   1:  PR[GP1:91,1] = PR[GP1:90,1] + 38.057;
   1:  PR[GP1:91,2] = PR[GP1:90,2] + -35.573;
   1:L PR[91] 10mm/sec CNT100;
   1:  PR[GP1:91,1] = PR[GP1:90,1] + 42.822;
   1:  PR[GP1:91,2] = PR[GP1:90,2] + -33.695;
   1:L PR[91] 10mm/sec CNT100;
   1:  PR[GP1:91,1] = PR[GP1:90,1] + 46.775;
   1:  PR[GP1:91,2] = PR[GP1:90,2] + -32.295;
   1:L PR[91] 10mm/sec CNT100;
   1:  PR[GP1:91,1] = PR[GP1:90,1] + 51.154;
   1:  PR[GP1:91,2] = PR[GP1:90,2] + -29.580;
   1:L PR[91] 10mm/sec CNT100;
   1:  PR[GP1:91,1] = PR[GP1:90,1] + 55.415;
   1:  PR[GP1:91,2] = PR[GP1:90,2] + -25.807;
   1:L PR[91] 10mm/sec CNT100;
   1:  PR[GP1:91,1] = PR[GP1:90,1] + 57.463;
   1:  PR[GP1:91,2] = PR[GP1:90,2] + -24.149;
   1:L PR[91] 10mm/sec CNT100;
   1:  PR[GP1:91,1] = PR[GP1:90,1] + 60.946;
   1:  PR[GP1:91,2] = PR[GP1:90,2] + -19.628;
   1:L PR[91] 10mm/sec CNT100;
   1:  PR[GP1:91,1] = PR[GP1:90,1] + 63.849;
   1:  PR[GP1:91,2] = PR[GP1:90,2] + -14.057;
   1:L PR[91] 10mm/sec CNT100;
   1:  PR[GP1:91,1] = PR[GP1:90,1] + 64.641;
   1:  PR[GP1:91,2] = PR[GP1:90,2] + -12.738;
   1:L PR[91] 10mm/sec CNT100;
   1:  PR[GP1:91,1] = PR[GP1:90,1] + 66.291;
   1:  PR[GP1:91,2] = PR[GP1:90,2] + -7.215;
   1:L PR[91] 10mm/sec CNT100;
   1:  PR[GP1:91,1] = PR[GP1:90,1] + 66.863;
   1:  PR[GP1:91,2] = PR[GP1:90,2] + -1.098;
   1:L PR[91] 10mm/sec CNT100;
   1:  PR[GP1:91,1] = PR[GP1:90,1] + 67.069;
   1:  PR[GP1:91,2] = PR[GP1:90,2] + 0.023;
   1:L PR[91] 10mm/sec CNT100;
   1:  PR[GP1:91,1] = PR[GP1:90,1] + 66.517;
   1:  PR[GP1:91,2] = PR[GP1:90,2] + 6.002;
   1:L PR[91] 10mm/sec CNT100;
   1:  PR[GP1:91,1] = PR[GP1:90,1] + 66.299;
   1:  PR[GP1:91,2] = PR[GP1:90,2] + 7.180;
   1:L PR[91] 10mm/sec CNT100;
   1:  PR[GP1:91,1] = PR[GP1:90,1] + 64.636;
   1:  PR[GP1:91,2] = PR[GP1:90,2] + 12.747;
   1:L PR[91] 10mm/sec CNT100;
   1:  PR[GP1:91,1] = PR[GP1:90,1] + 61.933;
   1:  PR[GP1:91,2] = PR[GP1:90,2] + 17.984;
   1:L PR[91] 10mm/sec CNT100;
   1:  PR[GP1:91,1] = PR[GP1:90,1] + 60.958;
   1:  PR[GP1:91,2] = PR[GP1:90,2] + 19.603;
   1:L PR[91] 10mm/sec CNT100;
   1:  PR[GP1:91,1] = PR[GP1:90,1] + 57.455;
   1:  PR[GP1:91,2] = PR[GP1:90,2] + 24.151;
   1:L PR[91] 10mm/sec CNT100;
   1:  PR[GP1:91,1] = PR[GP1:90,1] + 53.581;
   1:  PR[GP1:91,2] = PR[GP1:90,2] + 27.615;
   1:L PR[91] 10mm/sec CNT100;
   1:  PR[GP1:91,1] = PR[GP1:90,1] + 51.169;
   1:  PR[GP1:91,2] = PR[GP1:90,2] + 29.562;
   1:L PR[91] 10mm/sec CNT100;
   1:  PR[GP1:91,1] = PR[GP1:90,1] + 46.768;
   1:  PR[GP1:91,2] = PR[GP1:90,2] + 32.290;
   1:L PR[91] 10mm/sec CNT100;
   1:  PR[GP1:91,1] = PR[GP1:90,1] + 42.433;
   1:  PR[GP1:91,2] = PR[GP1:90,2] + 34.022;
   1:L PR[91] 10mm/sec CNT100;
   1:  PR[GP1:91,1] = PR[GP1:90,1] + 38.074;
   1:  PR[GP1:91,2] = PR[GP1:90,2] + 35.561;
   1:L PR[91] 10mm/sec CNT100;
   1:  PR[GP1:91,1] = PR[GP1:90,1] + 33.724;
   1:  PR[GP1:91,2] = PR[GP1:90,2] + 36.497;
   1:L PR[91] 10mm/sec CNT100;
   1:  PR[GP1:91,1] = PR[GP1:90,1] + 29.795;
   1:  PR[GP1:91,2] = PR[GP1:90,2] + 36.645;
   1:L PR[91] 10mm/sec CNT100;
   1:  PR[GP1:91,1] = PR[GP1:90,1] + 23.624;
   1:  PR[GP1:91,2] = PR[GP1:90,2] + 36.667;
   1:L PR[91] 10mm/sec CNT100;
   1:  PR[GP1:91,1] = PR[GP1:90,1] + 20.005;
   1:  PR[GP1:91,2] = PR[GP1:90,2] + 36.191;
   1:L PR[91] 10mm/sec CNT100;
   1:  PR[GP1:91,1] = PR[GP1:90,1] + 16.894;
   1:  PR[GP1:91,2] = PR[GP1:90,2] + 35.201;
   1:L PR[91] 10mm/sec CNT100;
   1:  PR[GP1:91,1] = PR[GP1:90,1] + 9.875;
   1:  PR[GP1:91,2] = PR[GP1:90,2] + 32.768;
   1:L PR[91] 10mm/sec CNT100;
   1:  PR[GP1:91,1] = PR[GP1:90,1] + 7.298;
   1:  PR[GP1:91,2] = PR[GP1:90,2] + 31.423;
   1:L PR[91] 10mm/sec CNT100;
   1:  PR[GP1:91,1] = PR[GP1:90,1] + 3.973;
   1:  PR[GP1:91,2] = PR[GP1:90,2] + 29.074;
   1:L PR[91] 10mm/sec CNT100;
   1:  PR[GP1:91,1] = PR[GP1:90,1] + 3.823;
   1:  PR[GP1:91,2] = PR[GP1:90,2] + 28.957;
   1:L PR[91] 10mm/sec CNT100;
   1:  PR[GP1:91,1] = PR[GP1:90,1] + 3.611;
   1:  PR[GP1:91,2] = PR[GP1:90,2] + 28.710;
   1:L PR[91] 10mm/sec CNT100;
   1:  PR[GP1:91,1] = PR[GP1:90,1] + 2.937;
   1:  PR[GP1:91,2] = PR[GP1:90,2] + 28.444;
   1:L PR[91] 10mm/sec CNT100;
   1:  PR[GP1:91,1] = PR[GP1:90,1] + 1.783;
   1:  PR[GP1:91,2] = PR[GP1:90,2] + 27.801;
   1:L PR[91] 10mm/sec CNT100;
   1:  PR[GP1:91,1] = PR[GP1:90,1] + 0.780;
   1:  PR[GP1:91,2] = PR[GP1:90,2] + 28.419;
   1:  PR[GP1:91,3] = PR[GP1:90,3] + 58.520;
   1:L PR[91] 10mm/sec CNT100;
   1:  PR[GP1:91,1] = PR[GP1:90,1] + -2.625;
   1:  PR[GP1:91,2] = PR[GP1:90,2] + 29.211;
   1:L PR[91] 10mm/sec CNT100;
   1:  PR[GP1:91,1] = PR[GP1:90,1] + -6.013;
   1:  PR[GP1:91,2] = PR[GP1:90,2] + 31.605;
   1:L PR[91] 10mm/sec CNT100;
   1:  PR[GP1:91,1] = PR[GP1:90,1] + -8.315;
   1:  PR[GP1:91,2] = PR[GP1:90,2] + 32.809;
   1:L PR[91] 10mm/sec CNT100;
   1:  PR[GP1:91,1] = PR[GP1:90,1] + -11.164;
   1:  PR[GP1:91,2] = PR[GP1:90,2] + 33.725;
   1:L PR[91] 10mm/sec CNT100;
   1:  PR[GP1:91,1] = PR[GP1:90,1] + -18.764;
   1:  PR[GP1:91,2] = PR[GP1:90,2] + 36.352;
   1:L PR[91] 10mm/sec CNT100;
   1:  PR[GP1:91,1] = PR[GP1:90,1] + -22.038;
   1:  PR[GP1:91,2] = PR[GP1:90,2] + 36.780;
   1:L PR[91] 10mm/sec CNT100;
   1:  PR[GP1:91,1] = PR[GP1:90,1] + -25.898;
   1:  PR[GP1:91,2] = PR[GP1:90,2] + 36.647;
   1:L PR[91] 10mm/sec CNT100;
   1:  PR[GP1:91,1] = PR[GP1:90,1] + -32.531;
   1:  PR[GP1:91,2] = PR[GP1:90,2] + 36.614;
   1:L PR[91] 10mm/sec CNT100;
   1:  PR[GP1:91,1] = PR[GP1:90,1] + -36.524;
   1:  PR[GP1:91,2] = PR[GP1:90,2] + 35.753;
   1:L PR[91] 10mm/sec CNT100;
   1:  PR[GP1:91,1] = PR[GP1:90,1] + -40.912;
   1:  PR[GP1:91,2] = PR[GP1:90,2] + 34.015;
   1:L PR[91] 10mm/sec CNT100;
   1:  PR[GP1:91,1] = PR[GP1:90,1] + -45.583;
   1:  PR[GP1:91,2] = PR[GP1:90,2] + 32.357;
   1:L PR[91] 10mm/sec CNT100;
   1:  PR[GP1:91,1] = PR[GP1:90,1] + -49.681;
   1:  PR[GP1:91,2] = PR[GP1:90,2] + 29.804;
   1:L PR[91] 10mm/sec CNT100;
   1:  PR[GP1:91,1] = PR[GP1:90,1] + -53.670;
   1:  PR[GP1:91,2] = PR[GP1:90,2] + 26.262;
   1:L PR[91] 10mm/sec CNT100;
   1:  PR[GP1:91,1] = PR[GP1:90,1] + -56.314;
   1:  PR[GP1:91,2] = PR[GP1:90,2] + 24.122;
   1:L PR[91] 10mm/sec CNT100;
   1:  PR[GP1:91,1] = PR[GP1:90,1] + -59.540;
   1:  PR[GP1:91,2] = PR[GP1:90,2] + 19.923;
   1:L PR[91] 10mm/sec CNT100;
   1:  PR[GP1:91,1] = PR[GP1:90,1] + -62.253;
   1:  PR[GP1:91,2] = PR[GP1:90,2] + 14.659;
   1:L PR[91] 10mm/sec CNT100;
   1:  PR[GP1:91,1] = PR[GP1:90,1] + -63.437;
   1:  PR[GP1:91,2] = PR[GP1:90,2] + 12.681;
   1:L PR[91] 10mm/sec CNT100;
   1:  PR[GP1:91,1] = PR[GP1:90,1] + -64.989;
   1:  PR[GP1:91,2] = PR[GP1:90,2] + 7.415;
   1:L PR[91] 10mm/sec CNT100;
   1:  PR[GP1:91,1] = PR[GP1:90,1] + -65.501;
   1:  PR[GP1:91,2] = PR[GP1:90,2] + 1.817;
   1:L PR[91] 10mm/sec CNT100;
   1:  PR[GP1:91,1] = PR[GP1:90,1] + -65.842;
   1:  PR[GP1:91,2] = PR[GP1:90,2] + -0.032;
   1:L PR[91] 10mm/sec CNT100;
   1:  PR[GP1:91,1] = PR[GP1:90,1] + -65.348;
   1:  PR[GP1:91,2] = PR[GP1:90,2] + -5.509;
   1:L PR[91] 10mm/sec CNT100;
   1:  PR[GP1:91,1] = PR[GP1:90,1] + -64.997;
   1:  PR[GP1:91,2] = PR[GP1:90,2] + -7.398;
   1:L PR[91] 10mm/sec CNT100;
   1:  PR[GP1:91,1] = PR[GP1:90,1] + -63.431;
   1:  PR[GP1:91,2] = PR[GP1:90,2] + -12.710;
   1:L PR[91] 10mm/sec CNT100;
   1:  PR[GP1:91,1] = PR[GP1:90,1] + -60.899;
   1:  PR[GP1:91,2] = PR[GP1:90,2] + -17.675;
   1:L PR[91] 10mm/sec CNT100;
   1:  PR[GP1:91,1] = PR[GP1:90,1] + -59.551;
   1:  PR[GP1:91,2] = PR[GP1:90,2] + -19.917;
   1:L PR[91] 10mm/sec CNT100;
   1:  PR[GP1:91,1] = PR[GP1:90,1] + -56.303;
   1:  PR[GP1:91,2] = PR[GP1:90,2] + -24.145;
   1:L PR[91] 10mm/sec CNT100;
   1:  PR[GP1:91,1] = PR[GP1:90,1] + -52.655;
   1:  PR[GP1:91,2] = PR[GP1:90,2] + -27.417;
   1:L PR[91] 10mm/sec CNT100;
   1:  PR[GP1:91,1] = PR[GP1:90,1] + -49.690;
   1:  PR[GP1:91,2] = PR[GP1:90,2] + -29.807;
   1:L PR[91] 10mm/sec CNT100;
   1:  PR[GP1:91,1] = PR[GP1:90,1] + -45.569;
   1:  PR[GP1:91,2] = PR[GP1:90,2] + -32.374;
   1:L PR[91] 10mm/sec CNT100;
   1:  PR[GP1:91,1] = PR[GP1:90,1] + -41.541;
   1:  PR[GP1:91,2] = PR[GP1:90,2] + -33.992;
   1:L PR[91] 10mm/sec CNT100;
   1:  PR[GP1:91,1] = PR[GP1:90,1] + -36.528;
   1:  PR[GP1:91,2] = PR[GP1:90,2] + -35.760;
   1:L PR[91] 10mm/sec CNT100;
   1:  PR[GP1:91,1] = PR[GP1:90,1] + -32.514;
   1:  PR[GP1:91,2] = PR[GP1:90,2] + -36.626;
   1:L PR[91] 10mm/sec CNT100;
   1:  PR[GP1:91,1] = PR[GP1:90,1] + -28.876;
   1:  PR[GP1:91,2] = PR[GP1:90,2] + -36.766;
   1:L PR[91] 10mm/sec CNT100;
   1:  PR[GP1:91,1] = PR[GP1:90,1] + -22.036;
   1:  PR[GP1:91,2] = PR[GP1:90,2] + -36.788;
   1:L PR[91] 10mm/sec CNT100;
   1:  PR[GP1:91,1] = PR[GP1:90,1] + -18.744;
   1:  PR[GP1:91,2] = PR[GP1:90,2] + -36.358;
   1:L PR[91] 10mm/sec CNT100;
   1:  PR[GP1:91,1] = PR[GP1:90,1] + -15.922;
   1:  PR[GP1:91,2] = PR[GP1:90,2] + -35.460;
   1:L PR[91] 10mm/sec CNT100;
   1:  PR[GP1:91,1] = PR[GP1:90,1] + -8.309;
   1:  PR[GP1:91,2] = PR[GP1:90,2] + -32.814;
   1:L PR[91] 10mm/sec CNT100;
   1:  PR[GP1:91,1] = PR[GP1:90,1] + -6.009;
   1:  PR[GP1:91,2] = PR[GP1:90,2] + -31.611;
   1:L PR[91] 10mm/sec CNT100;
   1:  PR[GP1:91,1] = PR[GP1:90,1] + -2.582;
   1:  PR[GP1:91,2] = PR[GP1:90,2] + -29.121;
   1:L PR[91] 10mm/sec CNT100;
   1:  PR[GP1:91,1] = PR[GP1:90,1] + -1.792;
   1:  PR[GP1:91,2] = PR[GP1:90,2] + -29.090;
   1:L PR[91] 10mm/sec CNT100;
   1:  PR[GP1:91,1] = PR[GP1:90,1] + 1.871;
   1:  PR[GP1:91,2] = PR[GP1:90,2] + -28.308;
   1:L PR[91] 10mm/sec CNT100;
   1:  PR[GP1:91,1] = PR[GP1:90,1] + 2.128;
   1:  PR[GP1:91,2] = PR[GP1:90,2] + -28.515;
   1:L PR[91] 10mm/sec CNT100;
   1:  PR[GP1:91,1] = PR[GP1:90,1] + 3.505;
   1:  PR[GP1:91,2] = PR[GP1:90,2] + -29.200;
   1:L PR[91] 10mm/sec CNT100;
   1:  PR[GP1:91,1] = PR[GP1:90,1] + 6.833;
   1:  PR[GP1:91,2] = PR[GP1:90,2] + -31.618;
   1:L PR[91] 10mm/sec CNT100;
   1:  PR[GP1:91,1] = PR[GP1:90,1] + 9.111;
   1:  PR[GP1:91,2] = PR[GP1:90,2] + -32.807;
   1:L PR[91] 10mm/sec CNT100;
   1:  PR[GP1:91,1] = PR[GP1:90,1] + 11.958;
   1:  PR[GP1:91,2] = PR[GP1:90,2] + -33.722;
   1:L PR[91] 10mm/sec CNT100;
   1:  PR[GP1:91,1] = PR[GP1:90,1] + 19.568;
   1:  PR[GP1:91,2] = PR[GP1:90,2] + -36.356;
   1:L PR[91] 10mm/sec CNT100;
   1:  PR[GP1:91,1] = PR[GP1:90,1] + 22.838;
   1:  PR[GP1:91,2] = PR[GP1:90,2] + -36.786;
   1:L PR[91] 10mm/sec CNT100;
   1:  PR[GP1:91,1] = PR[GP1:90,1] + 26.679;
   1:  PR[GP1:91,2] = PR[GP1:90,2] + -36.657;
   1:L PR[91] 10mm/sec CNT100;
   1:  PR[GP1:91,1] = PR[GP1:90,1] + 33.319;
   1:  PR[GP1:91,2] = PR[GP1:90,2] + -36.628;
   1:L PR[91] 10mm/sec CNT100;
   1:  PR[GP1:91,1] = PR[GP1:90,1] + 37.305;
   1:  PR[GP1:91,2] = PR[GP1:90,2] + -35.770;
   1:L PR[91] 10mm/sec CNT100;
   1:  PR[GP1:91,1] = PR[GP1:90,1] + 41.699;
   1:  PR[GP1:91,2] = PR[GP1:90,2] + -34.039;
   1:L PR[91] 10mm/sec CNT100;
   1:  PR[GP1:91,1] = PR[GP1:90,1] + 46.376;
   1:  PR[GP1:91,2] = PR[GP1:90,2] + -32.381;
   1:L PR[91] 10mm/sec CNT100;
   1:  PR[GP1:91,1] = PR[GP1:90,1] + 50.449;
   1:  PR[GP1:91,2] = PR[GP1:90,2] + -29.857;
   1:L PR[91] 10mm/sec CNT100;
   1:  PR[GP1:91,1] = PR[GP1:90,1] + 54.416;
   1:  PR[GP1:91,2] = PR[GP1:90,2] + -26.344;
   1:L PR[91] 10mm/sec CNT100;
   1:  PR[GP1:91,1] = PR[GP1:90,1] + 57.067;
   1:  PR[GP1:91,2] = PR[GP1:90,2] + -24.198;
   1:L PR[91] 10mm/sec CNT100;
   1:  PR[GP1:91,1] = PR[GP1:90,1] + 60.327;
   1:  PR[GP1:91,2] = PR[GP1:90,2] + -19.966;
   1:L PR[91] 10mm/sec CNT100;
   1:  PR[GP1:91,1] = PR[GP1:90,1] + 63.048;
   1:  PR[GP1:91,2] = PR[GP1:90,2] + -14.745;
   1:L PR[91] 10mm/sec CNT100;
   1:  PR[GP1:91,1] = PR[GP1:90,1] + 64.235;
   1:  PR[GP1:91,2] = PR[GP1:90,2] + -12.768;
   1:L PR[91] 10mm/sec CNT100;
   1:  PR[GP1:91,1] = PR[GP1:90,1] + 65.784;
   1:  PR[GP1:91,2] = PR[GP1:90,2] + -7.581;
   1:L PR[91] 10mm/sec CNT100;
   1:  PR[GP1:91,1] = PR[GP1:90,1] + 66.322;
   1:  PR[GP1:91,2] = PR[GP1:90,2] + -1.828;
   1:L PR[91] 10mm/sec CNT100;
   1:  PR[GP1:91,1] = PR[GP1:90,1] + 66.663;
   1:  PR[GP1:91,2] = PR[GP1:90,2] + 0.023;
   1:L PR[91] 10mm/sec CNT100;
   1:  PR[GP1:91,1] = PR[GP1:90,1] + 66.143;
   1:  PR[GP1:91,2] = PR[GP1:90,2] + 5.652;
   1:L PR[91] 10mm/sec CNT100;
   1:  PR[GP1:91,1] = PR[GP1:90,1] + 65.792;
   1:  PR[GP1:91,2] = PR[GP1:90,2] + 7.545;
   1:L PR[91] 10mm/sec CNT100;
   1:  PR[GP1:91,1] = PR[GP1:90,1] + 64.229;
   1:  PR[GP1:91,2] = PR[GP1:90,2] + 12.777;
   1:L PR[91] 10mm/sec CNT100;
   1:  PR[GP1:91,1] = PR[GP1:90,1] + 61.689;
   1:  PR[GP1:91,2] = PR[GP1:90,2] + 17.700;
   1:L PR[91] 10mm/sec CNT100;
   1:  PR[GP1:91,1] = PR[GP1:90,1] + 60.340;
   1:  PR[GP1:91,2] = PR[GP1:90,2] + 19.941;
   1:L PR[91] 10mm/sec CNT100;
   1:  PR[GP1:91,1] = PR[GP1:90,1] + 57.060;
   1:  PR[GP1:91,2] = PR[GP1:90,2] + 24.199;
   1:L PR[91] 10mm/sec CNT100;
   1:  PR[GP1:91,1] = PR[GP1:90,1] + 53.431;
   1:  PR[GP1:91,2] = PR[GP1:90,2] + 27.444;
   1:L PR[91] 10mm/sec CNT100;
   1:  PR[GP1:91,1] = PR[GP1:90,1] + 50.464;
   1:  PR[GP1:91,2] = PR[GP1:90,2] + 29.839;
   1:L PR[91] 10mm/sec CNT100;
   1:  PR[GP1:91,1] = PR[GP1:90,1] + 46.370;
   1:  PR[GP1:91,2] = PR[GP1:90,2] + 32.377;
   1:L PR[91] 10mm/sec CNT100;
   1:  PR[GP1:91,1] = PR[GP1:90,1] + 42.336;
   1:  PR[GP1:91,2] = PR[GP1:90,2] + 33.988;
   1:L PR[91] 10mm/sec CNT100;
   1:  PR[GP1:91,1] = PR[GP1:90,1] + 37.323;
   1:  PR[GP1:91,2] = PR[GP1:90,2] + 35.758;
   1:L PR[91] 10mm/sec CNT100;
   1:  PR[GP1:91,1] = PR[GP1:90,1] + 33.316;
   1:  PR[GP1:91,2] = PR[GP1:90,2] + 36.620;
   1:L PR[91] 10mm/sec CNT100;
   1:  PR[GP1:91,1] = PR[GP1:90,1] + 29.696;
   1:  PR[GP1:91,2] = PR[GP1:90,2] + 36.757;
   1:L PR[91] 10mm/sec CNT100;
   1:  PR[GP1:91,1] = PR[GP1:90,1] + 22.858;
   1:  PR[GP1:91,2] = PR[GP1:90,2] + 36.781;
   1:L PR[91] 10mm/sec CNT100;
   1:  PR[GP1:91,1] = PR[GP1:90,1] + 19.572;
   1:  PR[GP1:91,2] = PR[GP1:90,2] + 36.349;
   1:L PR[91] 10mm/sec CNT100;
   1:  PR[GP1:91,1] = PR[GP1:90,1] + 16.746;
   1:  PR[GP1:91,2] = PR[GP1:90,2] + 35.449;
   1:L PR[91] 10mm/sec CNT100;
   1:  PR[GP1:91,1] = PR[GP1:90,1] + 9.130;
   1:  PR[GP1:91,2] = PR[GP1:90,2] + 32.809;
   1:L PR[91] 10mm/sec CNT100;
   1:  PR[GP1:91,1] = PR[GP1:90,1] + 6.837;
   1:  PR[GP1:91,2] = PR[GP1:90,2] + 31.612;
   1:L PR[91] 10mm/sec CNT100;
   1:  PR[GP1:91,1] = PR[GP1:90,1] + 3.510;
   1:  PR[GP1:91,2] = PR[GP1:90,2] + 29.256;
   1:L PR[91] 10mm/sec CNT100;
   1:  PR[GP1:91,1] = PR[GP1:90,1] + 1.849;
   1:  PR[GP1:91,2] = PR[GP1:90,2] + 28.332;
   1:L PR[91] 10mm/sec CNT100;
   1:  PR[GP1:91,1] = PR[GP1:90,1] + 0.451;
   1:  PR[GP1:91,2] = PR[GP1:90,2] + 28.982;
   1:  PR[GP1:91,3] = PR[GP1:90,3] + 59.850;
   1:L PR[91] 10mm/sec CNT100;
   1:  PR[GP1:91,1] = PR[GP1:90,1] + -2.564;
   1:  PR[GP1:91,2] = PR[GP1:90,2] + 29.683;
   1:L PR[91] 10mm/sec CNT100;
   1:  PR[GP1:91,1] = PR[GP1:90,1] + -5.554;
   1:  PR[GP1:91,2] = PR[GP1:90,2] + 31.796;
   1:L PR[91] 10mm/sec CNT100;
   1:  PR[GP1:91,1] = PR[GP1:90,1] + -7.570;
   1:  PR[GP1:91,2] = PR[GP1:90,2] + 32.850;
   1:L PR[91] 10mm/sec CNT100;
   1:  PR[GP1:91,1] = PR[GP1:90,1] + -10.072;
   1:  PR[GP1:91,2] = PR[GP1:90,2] + 33.654;
   1:L PR[91] 10mm/sec CNT100;
   1:  PR[GP1:91,1] = PR[GP1:90,1] + -18.331;
   1:  PR[GP1:91,2] = PR[GP1:90,2] + 36.509;
   1:L PR[91] 10mm/sec CNT100;
   1:  PR[GP1:91,1] = PR[GP1:90,1] + -21.272;
   1:  PR[GP1:91,2] = PR[GP1:90,2] + 36.894;
   1:L PR[91] 10mm/sec CNT100;
   1:  PR[GP1:91,1] = PR[GP1:90,1] + -24.746;
   1:  PR[GP1:91,2] = PR[GP1:90,2] + 36.774;
   1:L PR[91] 10mm/sec CNT100;
   1:  PR[GP1:91,1] = PR[GP1:90,1] + -32.122;
   1:  PR[GP1:91,2] = PR[GP1:90,2] + 36.737;
   1:L PR[91] 10mm/sec CNT100;
   1:  PR[GP1:91,1] = PR[GP1:90,1] + -35.770;
   1:  PR[GP1:91,2] = PR[GP1:90,2] + 35.950;
   1:L PR[91] 10mm/sec CNT100;
   1:  PR[GP1:91,1] = PR[GP1:90,1] + -39.787;
   1:  PR[GP1:91,2] = PR[GP1:90,2] + 34.360;
   1:L PR[91] 10mm/sec CNT100;
   1:  PR[GP1:91,1] = PR[GP1:90,1] + -45.183;
   1:  PR[GP1:91,2] = PR[GP1:90,2] + 32.444;
   1:L PR[91] 10mm/sec CNT100;
   1:  PR[GP1:91,1] = PR[GP1:90,1] + -48.972;
   1:  PR[GP1:91,2] = PR[GP1:90,2] + 30.083;
   1:L PR[91] 10mm/sec CNT100;
   1:  PR[GP1:91,1] = PR[GP1:90,1] + -52.666;
   1:  PR[GP1:91,2] = PR[GP1:90,2] + 26.803;
   1:L PR[91] 10mm/sec CNT100;
   1:  PR[GP1:91,1] = PR[GP1:90,1] + -55.914;
   1:  PR[GP1:91,2] = PR[GP1:90,2] + 24.175;
   1:L PR[91] 10mm/sec CNT100;
   1:  PR[GP1:91,1] = PR[GP1:90,1] + -58.920;
   1:  PR[GP1:91,2] = PR[GP1:90,2] + 20.263;
   1:L PR[91] 10mm/sec CNT100;
   1:  PR[GP1:91,1] = PR[GP1:90,1] + -61.450;
   1:  PR[GP1:91,2] = PR[GP1:90,2] + 15.353;
   1:L PR[91] 10mm/sec CNT100;
   1:  PR[GP1:91,1] = PR[GP1:90,1] + -63.029;
   1:  PR[GP1:91,2] = PR[GP1:90,2] + 12.715;
   1:L PR[91] 10mm/sec CNT100;
   1:  PR[GP1:91,1] = PR[GP1:90,1] + -64.481;
   1:  PR[GP1:91,2] = PR[GP1:90,2] + 7.789;
   1:L PR[91] 10mm/sec CNT100;
   1:  PR[GP1:91,1] = PR[GP1:90,1] + -64.961;
   1:  PR[GP1:91,2] = PR[GP1:90,2] + 2.546;
   1:L PR[91] 10mm/sec CNT100;
   1:  PR[GP1:91,1] = PR[GP1:90,1] + -65.436;
   1:  PR[GP1:91,2] = PR[GP1:90,2] + -0.032;
   1:L PR[91] 10mm/sec CNT100;
   1:  PR[GP1:91,1] = PR[GP1:90,1] + -64.972;
   1:  PR[GP1:91,2] = PR[GP1:90,2] + -5.168;
   1:L PR[91] 10mm/sec CNT100;
   1:  PR[GP1:91,1] = PR[GP1:90,1] + -64.489;
   1:  PR[GP1:91,2] = PR[GP1:90,2] + -7.772;
   1:L PR[91] 10mm/sec CNT100;
   1:  PR[GP1:91,1] = PR[GP1:90,1] + -63.023;
   1:  PR[GP1:91,2] = PR[GP1:90,2] + -12.744;
   1:L PR[91] 10mm/sec CNT100;
   1:  PR[GP1:91,1] = PR[GP1:90,1] + -60.652;
   1:  PR[GP1:91,2] = PR[GP1:90,2] + -17.392;
   1:L PR[91] 10mm/sec CNT100;
   1:  PR[GP1:91,1] = PR[GP1:90,1] + -58.930;
   1:  PR[GP1:91,2] = PR[GP1:90,2] + -20.258;
   1:L PR[91] 10mm/sec CNT100;
   1:  PR[GP1:91,1] = PR[GP1:90,1] + -55.903;
   1:  PR[GP1:91,2] = PR[GP1:90,2] + -24.198;
   1:L PR[91] 10mm/sec CNT100;
   1:  PR[GP1:91,1] = PR[GP1:90,1] + -52.502;
   1:  PR[GP1:91,2] = PR[GP1:90,2] + -27.248;
   1:L PR[91] 10mm/sec CNT100;
   1:  PR[GP1:91,1] = PR[GP1:90,1] + -48.981;
   1:  PR[GP1:91,2] = PR[GP1:90,2] + -30.087;
   1:L PR[91] 10mm/sec CNT100;
   1:  PR[GP1:91,1] = PR[GP1:90,1] + -45.168;
   1:  PR[GP1:91,2] = PR[GP1:90,2] + -32.462;
   1:L PR[91] 10mm/sec CNT100;
   1:  PR[GP1:91,1] = PR[GP1:90,1] + -41.441;
   1:  PR[GP1:91,2] = PR[GP1:90,2] + -33.959;
   1:L PR[91] 10mm/sec CNT100;
   1:  PR[GP1:91,1] = PR[GP1:90,1] + -35.773;
   1:  PR[GP1:91,2] = PR[GP1:90,2] + -35.958;
   1:L PR[91] 10mm/sec CNT100;
   1:  PR[GP1:91,1] = PR[GP1:90,1] + -32.104;
   1:  PR[GP1:91,2] = PR[GP1:90,2] + -36.750;
   1:L PR[91] 10mm/sec CNT100;
   1:  PR[GP1:91,1] = PR[GP1:90,1] + -28.776;
   1:  PR[GP1:91,2] = PR[GP1:90,2] + -36.878;
   1:L PR[91] 10mm/sec CNT100;
   1:  PR[GP1:91,1] = PR[GP1:90,1] + -21.268;
   1:  PR[GP1:91,2] = PR[GP1:90,2] + -36.902;
   1:L PR[91] 10mm/sec CNT100;
   1:  PR[GP1:91,1] = PR[GP1:90,1] + -18.311;
   1:  PR[GP1:91,2] = PR[GP1:90,2] + -36.515;
   1:L PR[91] 10mm/sec CNT100;
   1:  PR[GP1:91,1] = PR[GP1:90,1] + -15.773;
   1:  PR[GP1:91,2] = PR[GP1:90,2] + -35.708;
   1:L PR[91] 10mm/sec CNT100;
   1:  PR[GP1:91,1] = PR[GP1:90,1] + -7.563;
   1:  PR[GP1:91,2] = PR[GP1:90,2] + -32.854;
   1:L PR[91] 10mm/sec CNT100;
   1:  PR[GP1:91,1] = PR[GP1:90,1] + -5.549;
   1:  PR[GP1:91,2] = PR[GP1:90,2] + -31.801;
   1:L PR[91] 10mm/sec CNT100;
   1:  PR[GP1:91,1] = PR[GP1:90,1] + -2.522;
   1:  PR[GP1:91,2] = PR[GP1:90,2] + -29.602;
   1:L PR[91] 10mm/sec CNT100;
   1:  PR[GP1:91,1] = PR[GP1:90,1] + -1.431;
   1:  PR[GP1:91,2] = PR[GP1:90,2] + -29.558;
   1:L PR[91] 10mm/sec CNT100;
   1:  PR[GP1:91,1] = PR[GP1:90,1] + 1.938;
   1:  PR[GP1:91,2] = PR[GP1:90,2] + -28.839;
   1:L PR[91] 10mm/sec CNT100;
   1:  PR[GP1:91,1] = PR[GP1:90,1] + 2.234;
   1:  PR[GP1:91,2] = PR[GP1:90,2] + -29.078;
   1:L PR[91] 10mm/sec CNT100;
   1:  PR[GP1:91,1] = PR[GP1:90,1] + 3.443;
   1:  PR[GP1:91,2] = PR[GP1:90,2] + -29.680;
   1:L PR[91] 10mm/sec CNT100;
   1:  PR[GP1:91,1] = PR[GP1:90,1] + 6.371;
   1:  PR[GP1:91,2] = PR[GP1:90,2] + -31.807;
   1:L PR[91] 10mm/sec CNT100;
   1:  PR[GP1:91,1] = PR[GP1:90,1] + 8.365;
   1:  PR[GP1:91,2] = PR[GP1:90,2] + -32.848;
   1:L PR[91] 10mm/sec CNT100;
   1:  PR[GP1:91,1] = PR[GP1:90,1] + 10.864;
   1:  PR[GP1:91,2] = PR[GP1:90,2] + -33.651;
   1:L PR[91] 10mm/sec CNT100;
   1:  PR[GP1:91,1] = PR[GP1:90,1] + 19.135;
   1:  PR[GP1:91,2] = PR[GP1:90,2] + -36.514;
   1:L PR[91] 10mm/sec CNT100;
   1:  PR[GP1:91,1] = PR[GP1:90,1] + 22.071;
   1:  PR[GP1:91,2] = PR[GP1:90,2] + -36.900;
   1:L PR[91] 10mm/sec CNT100;
   1:  PR[GP1:91,1] = PR[GP1:90,1] + 25.529;
   1:  PR[GP1:91,2] = PR[GP1:90,2] + -36.784;
   1:L PR[91] 10mm/sec CNT100;
   1:  PR[GP1:91,1] = PR[GP1:90,1] + 32.910;
   1:  PR[GP1:91,2] = PR[GP1:90,2] + -36.751;
   1:L PR[91] 10mm/sec CNT100;
   1:  PR[GP1:91,1] = PR[GP1:90,1] + 36.553;
   1:  PR[GP1:91,2] = PR[GP1:90,2] + -35.967;
   1:L PR[91] 10mm/sec CNT100;
   1:  PR[GP1:91,1] = PR[GP1:90,1] + 40.575;
   1:  PR[GP1:91,2] = PR[GP1:90,2] + -34.383;
   1:L PR[91] 10mm/sec CNT100;
   1:  PR[GP1:91,1] = PR[GP1:90,1] + 45.977;
   1:  PR[GP1:91,2] = PR[GP1:90,2] + -32.468;
   1:L PR[91] 10mm/sec CNT100;
   1:  PR[GP1:91,1] = PR[GP1:90,1] + 49.743;
   1:  PR[GP1:91,2] = PR[GP1:90,2] + -30.134;
   1:L PR[91] 10mm/sec CNT100;
   1:  PR[GP1:91,1] = PR[GP1:90,1] + 53.416;
   1:  PR[GP1:91,2] = PR[GP1:90,2] + -26.881;
   1:L PR[91] 10mm/sec CNT100;
   1:  PR[GP1:91,1] = PR[GP1:90,1] + 56.671;
   1:  PR[GP1:91,2] = PR[GP1:90,2] + -24.246;
   1:L PR[91] 10mm/sec CNT100;
   1:  PR[GP1:91,1] = PR[GP1:90,1] + 59.709;
   1:  PR[GP1:91,2] = PR[GP1:90,2] + -20.303;
   1:L PR[91] 10mm/sec CNT100;
   1:  PR[GP1:91,1] = PR[GP1:90,1] + 62.246;
   1:  PR[GP1:91,2] = PR[GP1:90,2] + -15.434;
   1:L PR[91] 10mm/sec CNT100;
   1:  PR[GP1:91,1] = PR[GP1:90,1] + 63.828;
   1:  PR[GP1:91,2] = PR[GP1:90,2] + -12.799;
   1:L PR[91] 10mm/sec CNT100;
   1:  PR[GP1:91,1] = PR[GP1:90,1] + 65.278;
   1:  PR[GP1:91,2] = PR[GP1:90,2] + -7.946;
   1:L PR[91] 10mm/sec CNT100;
   1:  PR[GP1:91,1] = PR[GP1:90,1] + 65.781;
   1:  PR[GP1:91,2] = PR[GP1:90,2] + -2.558;
   1:L PR[91] 10mm/sec CNT100;
   1:  PR[GP1:91,1] = PR[GP1:90,1] + 66.257;
   1:  PR[GP1:91,2] = PR[GP1:90,2] + 0.023;
   1:L PR[91] 10mm/sec CNT100;
   1:  PR[GP1:91,1] = PR[GP1:90,1] + 65.769;
   1:  PR[GP1:91,2] = PR[GP1:90,2] + 5.301;
   1:L PR[91] 10mm/sec CNT100;
   1:  PR[GP1:91,1] = PR[GP1:90,1] + 65.286;
   1:  PR[GP1:91,2] = PR[GP1:90,2] + 7.911;
   1:L PR[91] 10mm/sec CNT100;
   1:  PR[GP1:91,1] = PR[GP1:90,1] + 63.823;
   1:  PR[GP1:91,2] = PR[GP1:90,2] + 12.808;
   1:L PR[91] 10mm/sec CNT100;
   1:  PR[GP1:91,1] = PR[GP1:90,1] + 61.445;
   1:  PR[GP1:91,2] = PR[GP1:90,2] + 17.415;
   1:L PR[91] 10mm/sec CNT100;
   1:  PR[GP1:91,1] = PR[GP1:90,1] + 59.722;
   1:  PR[GP1:91,2] = PR[GP1:90,2] + 20.278;
   1:L PR[91] 10mm/sec CNT100;
   1:  PR[GP1:91,1] = PR[GP1:90,1] + 56.664;
   1:  PR[GP1:91,2] = PR[GP1:90,2] + 24.247;
   1:L PR[91] 10mm/sec CNT100;
   1:  PR[GP1:91,1] = PR[GP1:90,1] + 53.282;
   1:  PR[GP1:91,2] = PR[GP1:90,2] + 27.272;
   1:L PR[91] 10mm/sec CNT100;
   1:  PR[GP1:91,1] = PR[GP1:90,1] + 49.759;
   1:  PR[GP1:91,2] = PR[GP1:90,2] + 30.116;
   1:L PR[91] 10mm/sec CNT100;
   1:  PR[GP1:91,1] = PR[GP1:90,1] + 45.971;
   1:  PR[GP1:91,2] = PR[GP1:90,2] + 32.463;
   1:L PR[91] 10mm/sec CNT100;
   1:  PR[GP1:91,1] = PR[GP1:90,1] + 42.239;
   1:  PR[GP1:91,2] = PR[GP1:90,2] + 33.954;
   1:L PR[91] 10mm/sec CNT100;
   1:  PR[GP1:91,1] = PR[GP1:90,1] + 36.572;
   1:  PR[GP1:91,2] = PR[GP1:90,2] + 35.955;
   1:L PR[91] 10mm/sec CNT100;
   1:  PR[GP1:91,1] = PR[GP1:90,1] + 32.909;
   1:  PR[GP1:91,2] = PR[GP1:90,2] + 36.743;
   1:L PR[91] 10mm/sec CNT100;
   1:  PR[GP1:91,1] = PR[GP1:90,1] + 29.598;
   1:  PR[GP1:91,2] = PR[GP1:90,2] + 36.868;
   1:L PR[91] 10mm/sec CNT100;
   1:  PR[GP1:91,1] = PR[GP1:90,1] + 22.092;
   1:  PR[GP1:91,2] = PR[GP1:90,2] + 36.894;
   1:L PR[91] 10mm/sec CNT100;
   1:  PR[GP1:91,1] = PR[GP1:90,1] + 19.140;
   1:  PR[GP1:91,2] = PR[GP1:90,2] + 36.506;
   1:L PR[91] 10mm/sec CNT100;
   1:  PR[GP1:91,1] = PR[GP1:90,1] + 16.598;
   1:  PR[GP1:91,2] = PR[GP1:90,2] + 35.698;
   1:L PR[91] 10mm/sec CNT100;
   1:  PR[GP1:91,1] = PR[GP1:90,1] + 8.385;
   1:  PR[GP1:91,2] = PR[GP1:90,2] + 32.850;
   1:L PR[91] 10mm/sec CNT100;
   1:  PR[GP1:91,1] = PR[GP1:90,1] + 6.376;
   1:  PR[GP1:91,2] = PR[GP1:90,2] + 31.802;
   1:L PR[91] 10mm/sec CNT100;
   1:  PR[GP1:91,1] = PR[GP1:90,1] + 3.745;
   1:  PR[GP1:91,2] = PR[GP1:90,2] + 29.943;
   1:L PR[91] 10mm/sec CNT100;
   1:  PR[GP1:91,1] = PR[GP1:90,1] + 3.748;
   1:  PR[GP1:91,2] = PR[GP1:90,2] + 29.883;
   1:L PR[91] 10mm/sec CNT100;
   1:  PR[GP1:91,1] = PR[GP1:90,1] + 1.914;
   1:  PR[GP1:91,2] = PR[GP1:90,2] + 28.862;
   1:L PR[91] 10mm/sec CNT100;
   1:  PR[GP1:91,1] = PR[GP1:90,1] + 0.122;
   1:  PR[GP1:91,2] = PR[GP1:90,2] + 29.545;
   1:  PR[GP1:91,3] = PR[GP1:90,3] + 61.180;
   1:L PR[91] 10mm/sec CNT100;
   1:  PR[GP1:91,1] = PR[GP1:90,1] + -2.504;
   1:  PR[GP1:91,2] = PR[GP1:90,2] + 30.155;
   1:L PR[91] 10mm/sec CNT100;
   1:  PR[GP1:91,1] = PR[GP1:90,1] + -5.095;
   1:  PR[GP1:91,2] = PR[GP1:90,2] + 31.986;
   1:L PR[91] 10mm/sec CNT100;
   1:  PR[GP1:91,1] = PR[GP1:90,1] + -6.825;
   1:  PR[GP1:91,2] = PR[GP1:90,2] + 32.891;
   1:L PR[91] 10mm/sec CNT100;
   1:  PR[GP1:91,1] = PR[GP1:90,1] + -8.980;
   1:  PR[GP1:91,2] = PR[GP1:90,2] + 33.584;
   1:L PR[91] 10mm/sec CNT100;
   1:  PR[GP1:91,1] = PR[GP1:90,1] + -17.898;
   1:  PR[GP1:91,2] = PR[GP1:90,2] + 36.667;
   1:L PR[91] 10mm/sec CNT100;
   1:  PR[GP1:91,1] = PR[GP1:90,1] + -20.505;
   1:  PR[GP1:91,2] = PR[GP1:90,2] + 37.008;
   1:L PR[91] 10mm/sec CNT100;
   1:  PR[GP1:91,1] = PR[GP1:90,1] + -23.595;
   1:  PR[GP1:91,2] = PR[GP1:90,2] + 36.901;
   1:L PR[91] 10mm/sec CNT100;
   1:  PR[GP1:91,1] = PR[GP1:90,1] + -31.713;
   1:  PR[GP1:91,2] = PR[GP1:90,2] + 36.861;
   1:L PR[91] 10mm/sec CNT100;
   1:  PR[GP1:91,1] = PR[GP1:90,1] + -35.017;
   1:  PR[GP1:91,2] = PR[GP1:90,2] + 36.148;
   1:L PR[91] 10mm/sec CNT100;
   1:  PR[GP1:91,1] = PR[GP1:90,1] + -38.662;
   1:  PR[GP1:91,2] = PR[GP1:90,2] + 34.705;
   1:L PR[91] 10mm/sec CNT100;
   1:  PR[GP1:91,1] = PR[GP1:90,1] + -44.783;
   1:  PR[GP1:91,2] = PR[GP1:90,2] + 32.531;
   1:L PR[91] 10mm/sec CNT100;
   1:  PR[GP1:91,1] = PR[GP1:90,1] + -48.264;
   1:  PR[GP1:91,2] = PR[GP1:90,2] + 30.363;
   1:L PR[91] 10mm/sec CNT100;
   1:  PR[GP1:91,1] = PR[GP1:90,1] + -51.662;
   1:  PR[GP1:91,2] = PR[GP1:90,2] + 27.345;
   1:L PR[91] 10mm/sec CNT100;
   1:  PR[GP1:91,1] = PR[GP1:90,1] + -55.514;
   1:  PR[GP1:91,2] = PR[GP1:90,2] + 24.228;
   1:L PR[91] 10mm/sec CNT100;
   1:  PR[GP1:91,1] = PR[GP1:90,1] + -58.299;
   1:  PR[GP1:91,2] = PR[GP1:90,2] + 20.603;
   1:L PR[91] 10mm/sec CNT100;
   1:  PR[GP1:91,1] = PR[GP1:90,1] + -60.647;
   1:  PR[GP1:91,2] = PR[GP1:90,2] + 16.047;
   1:L PR[91] 10mm/sec CNT100;
   1:  PR[GP1:91,1] = PR[GP1:90,1] + -62.621;
   1:  PR[GP1:91,2] = PR[GP1:90,2] + 12.749;
   1:L PR[91] 10mm/sec CNT100;
   1:  PR[GP1:91,1] = PR[GP1:90,1] + -63.973;
   1:  PR[GP1:91,2] = PR[GP1:90,2] + 8.163;
   1:L PR[91] 10mm/sec CNT100;
   1:  PR[GP1:91,1] = PR[GP1:90,1] + -64.420;
   1:  PR[GP1:91,2] = PR[GP1:90,2] + 3.275;
   1:L PR[91] 10mm/sec CNT100;
   1:  PR[GP1:91,1] = PR[GP1:90,1] + -65.030;
   1:  PR[GP1:91,2] = PR[GP1:90,2] + -0.032;
   1:L PR[91] 10mm/sec CNT100;
   1:  PR[GP1:91,1] = PR[GP1:90,1] + -64.597;
   1:  PR[GP1:91,2] = PR[GP1:90,2] + -4.827;
   1:L PR[91] 10mm/sec CNT100;
   1:  PR[GP1:91,1] = PR[GP1:90,1] + -63.980;
   1:  PR[GP1:91,2] = PR[GP1:90,2] + -8.147;
   1:L PR[91] 10mm/sec CNT100;
   1:  PR[GP1:91,1] = PR[GP1:90,1] + -62.615;
   1:  PR[GP1:91,2] = PR[GP1:90,2] + -12.779;
   1:L PR[91] 10mm/sec CNT100;
   1:  PR[GP1:91,1] = PR[GP1:90,1] + -60.406;
   1:  PR[GP1:91,2] = PR[GP1:90,2] + -17.109;
   1:L PR[91] 10mm/sec CNT100;
   1:  PR[GP1:91,1] = PR[GP1:90,1] + -58.309;
   1:  PR[GP1:91,2] = PR[GP1:90,2] + -20.598;
   1:L PR[91] 10mm/sec CNT100;
   1:  PR[GP1:91,1] = PR[GP1:90,1] + -55.503;
   1:  PR[GP1:91,2] = PR[GP1:90,2] + -24.251;
   1:L PR[91] 10mm/sec CNT100;
   1:  PR[GP1:91,1] = PR[GP1:90,1] + -52.349;
   1:  PR[GP1:91,2] = PR[GP1:90,2] + -27.080;
   1:L PR[91] 10mm/sec CNT100;
   1:  PR[GP1:91,1] = PR[GP1:90,1] + -48.272;
   1:  PR[GP1:91,2] = PR[GP1:90,2] + -30.367;
   1:L PR[91] 10mm/sec CNT100;
   1:  PR[GP1:91,1] = PR[GP1:90,1] + -44.768;
   1:  PR[GP1:91,2] = PR[GP1:90,2] + -32.549;
   1:L PR[91] 10mm/sec CNT100;
   1:  PR[GP1:91,1] = PR[GP1:90,1] + -41.341;
   1:  PR[GP1:91,2] = PR[GP1:90,2] + -33.925;
   1:L PR[91] 10mm/sec CNT100;
   1:  PR[GP1:91,1] = PR[GP1:90,1] + -35.019;
   1:  PR[GP1:91,2] = PR[GP1:90,2] + -36.156;
   1:L PR[91] 10mm/sec CNT100;
   1:  PR[GP1:91,1] = PR[GP1:90,1] + -31.693;
   1:  PR[GP1:91,2] = PR[GP1:90,2] + -36.873;
   1:L PR[91] 10mm/sec CNT100;
   1:  PR[GP1:91,1] = PR[GP1:90,1] + -28.676;
   1:  PR[GP1:91,2] = PR[GP1:90,2] + -36.990;
   1:L PR[91] 10mm/sec CNT100;
   1:  PR[GP1:91,1] = PR[GP1:90,1] + -20.500;
   1:  PR[GP1:91,2] = PR[GP1:90,2] + -37.015;
   1:L PR[91] 10mm/sec CNT100;
   1:  PR[GP1:91,1] = PR[GP1:90,1] + -17.877;
   1:  PR[GP1:91,2] = PR[GP1:90,2] + -36.673;
   1:L PR[91] 10mm/sec CNT100;
   1:  PR[GP1:91,1] = PR[GP1:90,1] + -15.624;
   1:  PR[GP1:91,2] = PR[GP1:90,2] + -35.955;
   1:L PR[91] 10mm/sec CNT100;
   1:  PR[GP1:91,1] = PR[GP1:90,1] + -6.816;
   1:  PR[GP1:91,2] = PR[GP1:90,2] + -32.895;
   1:L PR[91] 10mm/sec CNT100;
   1:  PR[GP1:91,1] = PR[GP1:90,1] + -5.089;
   1:  PR[GP1:91,2] = PR[GP1:90,2] + -31.991;
   1:L PR[91] 10mm/sec CNT100;
   1:  PR[GP1:91,1] = PR[GP1:90,1] + -2.461;
   1:  PR[GP1:91,2] = PR[GP1:90,2] + -30.082;
   1:L PR[91] 10mm/sec CNT100;
   1:  PR[GP1:91,1] = PR[GP1:90,1] + -1.069;
   1:  PR[GP1:91,2] = PR[GP1:90,2] + -30.026;
   1:L PR[91] 10mm/sec CNT100;
   1:  PR[GP1:91,1] = PR[GP1:90,1] + 2.004;
   1:  PR[GP1:91,2] = PR[GP1:90,2] + -29.370;
   1:L PR[91] 10mm/sec CNT100;
   1:  PR[GP1:91,1] = PR[GP1:90,1] + 2.340;
   1:  PR[GP1:91,2] = PR[GP1:90,2] + -29.641;
   1:L PR[91] 10mm/sec CNT100;
   1:  PR[GP1:91,1] = PR[GP1:90,1] + 3.382;
   1:  PR[GP1:91,2] = PR[GP1:90,2] + -30.160;
   1:L PR[91] 10mm/sec CNT100;
   1:  PR[GP1:91,1] = PR[GP1:90,1] + 5.910;
   1:  PR[GP1:91,2] = PR[GP1:90,2] + -31.996;
   1:L PR[91] 10mm/sec CNT100;
   1:  PR[GP1:91,1] = PR[GP1:90,1] + 7.620;
   1:  PR[GP1:91,2] = PR[GP1:90,2] + -32.888;
   1:L PR[91] 10mm/sec CNT100;
   1:  PR[GP1:91,1] = PR[GP1:90,1] + 9.771;
   1:  PR[GP1:91,2] = PR[GP1:90,2] + -33.580;
   1:L PR[91] 10mm/sec CNT100;
   1:  PR[GP1:91,1] = PR[GP1:90,1] + 18.701;
   1:  PR[GP1:91,2] = PR[GP1:90,2] + -36.671;
   1:L PR[91] 10mm/sec CNT100;
   1:  PR[GP1:91,1] = PR[GP1:90,1] + 21.304;
   1:  PR[GP1:91,2] = PR[GP1:90,2] + -37.014;
   1:L PR[91] 10mm/sec CNT100;
   1:  PR[GP1:91,1] = PR[GP1:90,1] + 24.379;
   1:  PR[GP1:91,2] = PR[GP1:90,2] + -36.910;
   1:L PR[91] 10mm/sec CNT100;
   1:  PR[GP1:91,1] = PR[GP1:90,1] + 32.502;
   1:  PR[GP1:91,2] = PR[GP1:90,2] + -36.875;
   1:L PR[91] 10mm/sec CNT100;
   1:  PR[GP1:91,1] = PR[GP1:90,1] + 35.801;
   1:  PR[GP1:91,2] = PR[GP1:90,2] + -36.165;
   1:L PR[91] 10mm/sec CNT100;
   1:  PR[GP1:91,1] = PR[GP1:90,1] + 39.451;
   1:  PR[GP1:91,2] = PR[GP1:90,2] + -34.726;
   1:L PR[91] 10mm/sec CNT100;
   1:  PR[GP1:91,1] = PR[GP1:90,1] + 45.578;
   1:  PR[GP1:91,2] = PR[GP1:90,2] + -32.555;
   1:L PR[91] 10mm/sec CNT100;
   1:  PR[GP1:91,1] = PR[GP1:90,1] + 49.038;
   1:  PR[GP1:91,2] = PR[GP1:90,2] + -30.411;
   1:L PR[91] 10mm/sec CNT100;
   1:  PR[GP1:91,1] = PR[GP1:90,1] + 52.417;
   1:  PR[GP1:91,2] = PR[GP1:90,2] + -27.418;
   1:L PR[91] 10mm/sec CNT100;
   1:  PR[GP1:91,1] = PR[GP1:90,1] + 56.276;
   1:  PR[GP1:91,2] = PR[GP1:90,2] + -24.295;
   1:L PR[91] 10mm/sec CNT100;
   1:  PR[GP1:91,1] = PR[GP1:90,1] + 59.090;
   1:  PR[GP1:91,2] = PR[GP1:90,2] + -20.641;
   1:L PR[91] 10mm/sec CNT100;
   1:  PR[GP1:91,1] = PR[GP1:90,1] + 61.445;
   1:  PR[GP1:91,2] = PR[GP1:90,2] + -16.122;
   1:L PR[91] 10mm/sec CNT100;
   1:  PR[GP1:91,1] = PR[GP1:90,1] + 63.422;
   1:  PR[GP1:91,2] = PR[GP1:90,2] + -12.829;
   1:L PR[91] 10mm/sec CNT100;
   1:  PR[GP1:91,1] = PR[GP1:90,1] + 64.771;
   1:  PR[GP1:91,2] = PR[GP1:90,2] + -8.312;
   1:L PR[91] 10mm/sec CNT100;
   1:  PR[GP1:91,1] = PR[GP1:90,1] + 65.241;
   1:  PR[GP1:91,2] = PR[GP1:90,2] + -3.289;
   1:L PR[91] 10mm/sec CNT100;
   1:  PR[GP1:91,1] = PR[GP1:90,1] + 65.850;
   1:  PR[GP1:91,2] = PR[GP1:90,2] + 0.023;
   1:L PR[91] 10mm/sec CNT100;
   1:  PR[GP1:91,1] = PR[GP1:90,1] + 65.396;
   1:  PR[GP1:91,2] = PR[GP1:90,2] + 4.951;
   1:L PR[91] 10mm/sec CNT100;
   1:  PR[GP1:91,1] = PR[GP1:90,1] + 64.779;
   1:  PR[GP1:91,2] = PR[GP1:90,2] + 8.276;
   1:L PR[91] 10mm/sec CNT100;
   1:  PR[GP1:91,1] = PR[GP1:90,1] + 63.416;
   1:  PR[GP1:91,2] = PR[GP1:90,2] + 12.838;
   1:L PR[91] 10mm/sec CNT100;
   1:  PR[GP1:91,1] = PR[GP1:90,1] + 61.201;
   1:  PR[GP1:91,2] = PR[GP1:90,2] + 17.131;
   1:L PR[91] 10mm/sec CNT100;
   1:  PR[GP1:91,1] = PR[GP1:90,1] + 59.103;
   1:  PR[GP1:91,2] = PR[GP1:90,2] + 20.615;
   1:L PR[91] 10mm/sec CNT100;
   1:  PR[GP1:91,1] = PR[GP1:90,1] + 56.268;
   1:  PR[GP1:91,2] = PR[GP1:90,2] + 24.296;
   1:L PR[91] 10mm/sec CNT100;
   1:  PR[GP1:91,1] = PR[GP1:90,1] + 53.132;
   1:  PR[GP1:91,2] = PR[GP1:90,2] + 27.100;
   1:L PR[91] 10mm/sec CNT100;
   1:  PR[GP1:91,1] = PR[GP1:90,1] + 49.054;
   1:  PR[GP1:91,2] = PR[GP1:90,2] + 30.392;
   1:L PR[91] 10mm/sec CNT100;
   1:  PR[GP1:91,1] = PR[GP1:90,1] + 45.573;
   1:  PR[GP1:91,2] = PR[GP1:90,2] + 32.550;
   1:L PR[91] 10mm/sec CNT100;
   1:  PR[GP1:91,1] = PR[GP1:90,1] + 42.142;
   1:  PR[GP1:91,2] = PR[GP1:90,2] + 33.920;
   1:L PR[91] 10mm/sec CNT100;
   1:  PR[GP1:91,1] = PR[GP1:90,1] + 35.821;
   1:  PR[GP1:91,2] = PR[GP1:90,2] + 36.152;
   1:L PR[91] 10mm/sec CNT100;
   1:  PR[GP1:91,1] = PR[GP1:90,1] + 32.501;
   1:  PR[GP1:91,2] = PR[GP1:90,2] + 36.866;
   1:L PR[91] 10mm/sec CNT100;
   1:  PR[GP1:91,1] = PR[GP1:90,1] + 29.499;
   1:  PR[GP1:91,2] = PR[GP1:90,2] + 36.979;
   1:L PR[91] 10mm/sec CNT100;
   1:  PR[GP1:91,1] = PR[GP1:90,1] + 21.326;
   1:  PR[GP1:91,2] = PR[GP1:90,2] + 37.008;
   1:L PR[91] 10mm/sec CNT100;
   1:  PR[GP1:91,1] = PR[GP1:90,1] + 18.707;
   1:  PR[GP1:91,2] = PR[GP1:90,2] + 36.664;
   1:L PR[91] 10mm/sec CNT100;
   1:  PR[GP1:91,1] = PR[GP1:90,1] + 16.451;
   1:  PR[GP1:91,2] = PR[GP1:90,2] + 35.946;
   1:L PR[91] 10mm/sec CNT100;
   1:  PR[GP1:91,1] = PR[GP1:90,1] + 7.640;
   1:  PR[GP1:91,2] = PR[GP1:90,2] + 32.891;
   1:L PR[91] 10mm/sec CNT100;
   1:  PR[GP1:91,1] = PR[GP1:90,1] + 5.915;
   1:  PR[GP1:91,2] = PR[GP1:90,2] + 31.991;
   1:L PR[91] 10mm/sec CNT100;
   1:  PR[GP1:91,1] = PR[GP1:90,1] + 3.684;
   1:  PR[GP1:91,2] = PR[GP1:90,2] + 30.415;
   1:L PR[91] 10mm/sec CNT100;
   1:  PR[GP1:91,1] = PR[GP1:90,1] + 3.688;
   1:  PR[GP1:91,2] = PR[GP1:90,2] + 30.343;
   1:L PR[91] 10mm/sec CNT100;
   1:  PR[GP1:91,1] = PR[GP1:90,1] + 1.980;
   1:  PR[GP1:91,2] = PR[GP1:90,2] + 29.392;
   1:L PR[91] 10mm/sec CNT100;
   1:  PR[GP1:91,1] = PR[GP1:90,1] + -0.206;
   1:  PR[GP1:91,2] = PR[GP1:90,2] + 30.108;
   1:  PR[GP1:91,3] = PR[GP1:90,3] + 62.510;
   1:L PR[91] 10mm/sec CNT100;
   1:  PR[GP1:91,1] = PR[GP1:90,1] + -2.443;
   1:  PR[GP1:91,2] = PR[GP1:90,2] + 30.628;
   1:L PR[91] 10mm/sec CNT100;
   1:  PR[GP1:91,1] = PR[GP1:90,1] + -4.635;
   1:  PR[GP1:91,2] = PR[GP1:90,2] + 32.176;
   1:L PR[91] 10mm/sec CNT100;
   1:  PR[GP1:91,1] = PR[GP1:90,1] + -6.080;
   1:  PR[GP1:91,2] = PR[GP1:90,2] + 32.932;
   1:L PR[91] 10mm/sec CNT100;
   1:  PR[GP1:91,1] = PR[GP1:90,1] + -7.888;
   1:  PR[GP1:91,2] = PR[GP1:90,2] + 33.513;
   1:L PR[91] 10mm/sec CNT100;
   1:  PR[GP1:91,1] = PR[GP1:90,1] + -17.466;
   1:  PR[GP1:91,2] = PR[GP1:90,2] + 36.824;
   1:L PR[91] 10mm/sec CNT100;
   1:  PR[GP1:91,1] = PR[GP1:90,1] + -19.738;
   1:  PR[GP1:91,2] = PR[GP1:90,2] + 37.121;
   1:L PR[91] 10mm/sec CNT100;
   1:  PR[GP1:91,1] = PR[GP1:90,1] + -22.443;
   1:  PR[GP1:91,2] = PR[GP1:90,2] + 37.028;
   1:L PR[91] 10mm/sec CNT100;
   1:  PR[GP1:91,1] = PR[GP1:90,1] + -31.303;
   1:  PR[GP1:91,2] = PR[GP1:90,2] + 36.984;
   1:L PR[91] 10mm/sec CNT100;
   1:  PR[GP1:91,1] = PR[GP1:90,1] + -34.263;
   1:  PR[GP1:91,2] = PR[GP1:90,2] + 36.345;
   1:L PR[91] 10mm/sec CNT100;
   1:  PR[GP1:91,1] = PR[GP1:90,1] + -37.538;
   1:  PR[GP1:91,2] = PR[GP1:90,2] + 35.049;
   1:L PR[91] 10mm/sec CNT100;
   1:  PR[GP1:91,1] = PR[GP1:90,1] + -44.383;
   1:  PR[GP1:91,2] = PR[GP1:90,2] + 32.618;
   1:L PR[91] 10mm/sec CNT100;
   1:  PR[GP1:91,1] = PR[GP1:90,1] + -47.556;
   1:  PR[GP1:91,2] = PR[GP1:90,2] + 30.642;
   1:L PR[91] 10mm/sec CNT100;
   1:  PR[GP1:91,1] = PR[GP1:90,1] + -50.659;
   1:  PR[GP1:91,2] = PR[GP1:90,2] + 27.887;
   1:L PR[91] 10mm/sec CNT100;
   1:  PR[GP1:91,1] = PR[GP1:90,1] + -55.114;
   1:  PR[GP1:91,2] = PR[GP1:90,2] + 24.281;
   1:L PR[91] 10mm/sec CNT100;
   1:  PR[GP1:91,1] = PR[GP1:90,1] + -57.679;
   1:  PR[GP1:91,2] = PR[GP1:90,2] + 20.943;
   1:L PR[91] 10mm/sec CNT100;
   1:  PR[GP1:91,1] = PR[GP1:90,1] + -59.844;
   1:  PR[GP1:91,2] = PR[GP1:90,2] + 16.740;
   1:L PR[91] 10mm/sec CNT100;
   1:  PR[GP1:91,1] = PR[GP1:90,1] + -62.214;
   1:  PR[GP1:91,2] = PR[GP1:90,2] + 12.783;
   1:L PR[91] 10mm/sec CNT100;
   1:  PR[GP1:91,1] = PR[GP1:90,1] + -63.465;
   1:  PR[GP1:91,2] = PR[GP1:90,2] + 8.538;
   1:L PR[91] 10mm/sec CNT100;
   1:  PR[GP1:91,1] = PR[GP1:90,1] + -63.880;
   1:  PR[GP1:91,2] = PR[GP1:90,2] + 4.004;
   1:L PR[91] 10mm/sec CNT100;
   1:  PR[GP1:91,1] = PR[GP1:90,1] + -64.624;
   1:  PR[GP1:91,2] = PR[GP1:90,2] + -0.032;
   1:L PR[91] 10mm/sec CNT100;
   1:  PR[GP1:91,1] = PR[GP1:90,1] + -64.221;
   1:  PR[GP1:91,2] = PR[GP1:90,2] + -4.486;
   1:L PR[91] 10mm/sec CNT100;
   1:  PR[GP1:91,1] = PR[GP1:90,1] + -63.472;
   1:  PR[GP1:91,2] = PR[GP1:90,2] + -8.521;
   1:L PR[91] 10mm/sec CNT100;
   1:  PR[GP1:91,1] = PR[GP1:90,1] + -62.207;
   1:  PR[GP1:91,2] = PR[GP1:90,2] + -12.813;
   1:L PR[91] 10mm/sec CNT100;
   1:  PR[GP1:91,1] = PR[GP1:90,1] + -60.160;
   1:  PR[GP1:91,2] = PR[GP1:90,2] + -16.826;
   1:L PR[91] 10mm/sec CNT100;
   1:  PR[GP1:91,1] = PR[GP1:90,1] + -57.689;
   1:  PR[GP1:91,2] = PR[GP1:90,2] + -20.939;
   1:L PR[91] 10mm/sec CNT100;
   1:  PR[GP1:91,1] = PR[GP1:90,1] + -55.103;
   1:  PR[GP1:91,2] = PR[GP1:90,2] + -24.305;
   1:L PR[91] 10mm/sec CNT100;
   1:  PR[GP1:91,1] = PR[GP1:90,1] + -52.196;
   1:  PR[GP1:91,2] = PR[GP1:90,2] + -26.911;
   1:L PR[91] 10mm/sec CNT100;
   1:  PR[GP1:91,1] = PR[GP1:90,1] + -47.562;
   1:  PR[GP1:91,2] = PR[GP1:90,2] + -30.646;
   1:L PR[91] 10mm/sec CNT100;
   1:  PR[GP1:91,1] = PR[GP1:90,1] + -44.367;
   1:  PR[GP1:91,2] = PR[GP1:90,2] + -32.637;
   1:L PR[91] 10mm/sec CNT100;
   1:  PR[GP1:91,1] = PR[GP1:90,1] + -41.241;
   1:  PR[GP1:91,2] = PR[GP1:90,2] + -33.892;
   1:L PR[91] 10mm/sec CNT100;
   1:  PR[GP1:91,1] = PR[GP1:90,1] + -34.264;
   1:  PR[GP1:91,2] = PR[GP1:90,2] + -36.354;
   1:L PR[91] 10mm/sec CNT100;
   1:  PR[GP1:91,1] = PR[GP1:90,1] + -31.283;
   1:  PR[GP1:91,2] = PR[GP1:90,2] + -36.997;
   1:L PR[91] 10mm/sec CNT100;
   1:  PR[GP1:91,1] = PR[GP1:90,1] + -28.576;
   1:  PR[GP1:91,2] = PR[GP1:90,2] + -37.101;
   1:L PR[91] 10mm/sec CNT100;
   1:  PR[GP1:91,1] = PR[GP1:90,1] + -19.733;
   1:  PR[GP1:91,2] = PR[GP1:90,2] + -37.129;
   1:L PR[91] 10mm/sec CNT100;
   1:  PR[GP1:91,1] = PR[GP1:90,1] + -17.444;
   1:  PR[GP1:91,2] = PR[GP1:90,2] + -36.830;
   1:L PR[91] 10mm/sec CNT100;
   1:  PR[GP1:91,1] = PR[GP1:90,1] + -15.474;
   1:  PR[GP1:91,2] = PR[GP1:90,2] + -36.203;
   1:L PR[91] 10mm/sec CNT100;
   1:  PR[GP1:91,1] = PR[GP1:90,1] + -6.070;
   1:  PR[GP1:91,2] = PR[GP1:90,2] + -32.935;
   1:L PR[91] 10mm/sec CNT100;
   1:  PR[GP1:91,1] = PR[GP1:90,1] + -4.629;
   1:  PR[GP1:91,2] = PR[GP1:90,2] + -32.181;
   1:L PR[91] 10mm/sec CNT100;
   1:  PR[GP1:91,1] = PR[GP1:90,1] + -2.400;
   1:  PR[GP1:91,2] = PR[GP1:90,2] + -30.562;
   1:L PR[91] 10mm/sec CNT100;
   1:  PR[GP1:91,1] = PR[GP1:90,1] + -0.708;
   1:  PR[GP1:91,2] = PR[GP1:90,2] + -30.494;
   1:L PR[91] 10mm/sec CNT100;
   1:  PR[GP1:91,1] = PR[GP1:90,1] + 2.070;
   1:  PR[GP1:91,2] = PR[GP1:90,2] + -29.901;
   1:L PR[91] 10mm/sec CNT100;
   1:  PR[GP1:91,1] = PR[GP1:90,1] + 2.447;
   1:  PR[GP1:91,2] = PR[GP1:90,2] + -30.204;
   1:L PR[91] 10mm/sec CNT100;
   1:  PR[GP1:91,1] = PR[GP1:90,1] + 3.321;
   1:  PR[GP1:91,2] = PR[GP1:90,2] + -30.640;
   1:L PR[91] 10mm/sec CNT100;
   1:  PR[GP1:91,1] = PR[GP1:90,1] + 5.449;
   1:  PR[GP1:91,2] = PR[GP1:90,2] + -32.185;
   1:L PR[91] 10mm/sec CNT100;
   1:  PR[GP1:91,1] = PR[GP1:90,1] + 6.874;
   1:  PR[GP1:91,2] = PR[GP1:90,2] + -32.929;
   1:L PR[91] 10mm/sec CNT100;
   1:  PR[GP1:91,1] = PR[GP1:90,1] + 8.677;
   1:  PR[GP1:91,2] = PR[GP1:90,2] + -33.508;
   1:L PR[91] 10mm/sec CNT100;
   1:  PR[GP1:91,1] = PR[GP1:90,1] + 18.268;
   1:  PR[GP1:91,2] = PR[GP1:90,2] + -36.829;
   1:L PR[91] 10mm/sec CNT100;
   1:  PR[GP1:91,1] = PR[GP1:90,1] + 20.537;
   1:  PR[GP1:91,2] = PR[GP1:90,2] + -37.127;
   1:L PR[91] 10mm/sec CNT100;
   1:  PR[GP1:91,1] = PR[GP1:90,1] + 23.228;
   1:  PR[GP1:91,2] = PR[GP1:90,2] + -37.037;
   1:L PR[91] 10mm/sec CNT100;
   1:  PR[GP1:91,1] = PR[GP1:90,1] + 32.094;
   1:  PR[GP1:91,2] = PR[GP1:90,2] + -36.998;
   1:L PR[91] 10mm/sec CNT100;
   1:  PR[GP1:91,1] = PR[GP1:90,1] + 35.049;
   1:  PR[GP1:91,2] = PR[GP1:90,2] + -36.362;
   1:L PR[91] 10mm/sec CNT100;
   1:  PR[GP1:91,1] = PR[GP1:90,1] + 38.328;
   1:  PR[GP1:91,2] = PR[GP1:90,2] + -35.070;
   1:L PR[91] 10mm/sec CNT100;
   1:  PR[GP1:91,1] = PR[GP1:90,1] + 45.180;
   1:  PR[GP1:91,2] = PR[GP1:90,2] + -32.642;
   1:L PR[91] 10mm/sec CNT100;
   1:  PR[GP1:91,1] = PR[GP1:90,1] + 48.332;
   1:  PR[GP1:91,2] = PR[GP1:90,2] + -30.688;
   1:L PR[91] 10mm/sec CNT100;
   1:  PR[GP1:91,1] = PR[GP1:90,1] + 51.418;
   1:  PR[GP1:91,2] = PR[GP1:90,2] + -27.955;
   1:L PR[91] 10mm/sec CNT100;
   1:  PR[GP1:91,1] = PR[GP1:90,1] + 55.880;
   1:  PR[GP1:91,2] = PR[GP1:90,2] + -24.343;
   1:L PR[91] 10mm/sec CNT100;
   1:  PR[GP1:91,1] = PR[GP1:90,1] + 58.471;
   1:  PR[GP1:91,2] = PR[GP1:90,2] + -20.979;
   1:L PR[91] 10mm/sec CNT100;
   1:  PR[GP1:91,1] = PR[GP1:90,1] + 60.644;
   1:  PR[GP1:91,2] = PR[GP1:90,2] + -16.811;
   1:L PR[91] 10mm/sec CNT100;
   1:  PR[GP1:91,1] = PR[GP1:90,1] + 63.015;
   1:  PR[GP1:91,2] = PR[GP1:90,2] + -12.860;
   1:L PR[91] 10mm/sec CNT100;
   1:  PR[GP1:91,1] = PR[GP1:90,1] + 64.265;
   1:  PR[GP1:91,2] = PR[GP1:90,2] + -8.678;
   1:L PR[91] 10mm/sec CNT100;
   1:  PR[GP1:91,1] = PR[GP1:90,1] + 64.700;
   1:  PR[GP1:91,2] = PR[GP1:90,2] + -4.019;
   1:L PR[91] 10mm/sec CNT100;
   1:  PR[GP1:91,1] = PR[GP1:90,1] + 65.444;
   1:  PR[GP1:91,2] = PR[GP1:90,2] + 0.023;
   1:L PR[91] 10mm/sec CNT100;
   1:  PR[GP1:91,1] = PR[GP1:90,1] + 65.022;
   1:  PR[GP1:91,2] = PR[GP1:90,2] + 4.601;
   1:L PR[91] 10mm/sec CNT100;
   1:  PR[GP1:91,1] = PR[GP1:90,1] + 64.273;
   1:  PR[GP1:91,2] = PR[GP1:90,2] + 8.641;
   1:L PR[91] 10mm/sec CNT100;
   1:  PR[GP1:91,1] = PR[GP1:90,1] + 63.010;
   1:  PR[GP1:91,2] = PR[GP1:90,2] + 12.868;
   1:L PR[91] 10mm/sec CNT100;
   1:  PR[GP1:91,1] = PR[GP1:90,1] + 60.957;
   1:  PR[GP1:91,2] = PR[GP1:90,2] + 16.847;
   1:L PR[91] 10mm/sec CNT100;
   1:  PR[GP1:91,1] = PR[GP1:90,1] + 58.485;
   1:  PR[GP1:91,2] = PR[GP1:90,2] + 20.953;
   1:L PR[91] 10mm/sec CNT100;
   1:  PR[GP1:91,1] = PR[GP1:90,1] + 55.873;
   1:  PR[GP1:91,2] = PR[GP1:90,2] + 24.344;
   1:L PR[91] 10mm/sec CNT100;
   1:  PR[GP1:91,1] = PR[GP1:90,1] + 52.982;
   1:  PR[GP1:91,2] = PR[GP1:90,2] + 26.928;
   1:L PR[91] 10mm/sec CNT100;
   1:  PR[GP1:91,1] = PR[GP1:90,1] + 48.349;
   1:  PR[GP1:91,2] = PR[GP1:90,2] + 30.669;
   1:L PR[91] 10mm/sec CNT100;
   1:  PR[GP1:91,1] = PR[GP1:90,1] + 45.175;
   1:  PR[GP1:91,2] = PR[GP1:90,2] + 32.636;
   1:L PR[91] 10mm/sec CNT100;
   1:  PR[GP1:91,1] = PR[GP1:90,1] + 42.044;
   1:  PR[GP1:91,2] = PR[GP1:90,2] + 33.886;
   1:L PR[91] 10mm/sec CNT100;
   1:  PR[GP1:91,1] = PR[GP1:90,1] + 35.070;
   1:  PR[GP1:91,2] = PR[GP1:90,2] + 36.349;
   1:L PR[91] 10mm/sec CNT100;
   1:  PR[GP1:91,1] = PR[GP1:90,1] + 32.094;
   1:  PR[GP1:91,2] = PR[GP1:90,2] + 36.989;
   1:L PR[91] 10mm/sec CNT100;
   1:  PR[GP1:91,1] = PR[GP1:90,1] + 29.400;
   1:  PR[GP1:91,2] = PR[GP1:90,2] + 37.091;
   1:L PR[91] 10mm/sec CNT100;
   1:  PR[GP1:91,1] = PR[GP1:90,1] + 20.560;
   1:  PR[GP1:91,2] = PR[GP1:90,2] + 37.122;
   1:L PR[91] 10mm/sec CNT100;
   1:  PR[GP1:91,1] = PR[GP1:90,1] + 18.275;
   1:  PR[GP1:91,2] = PR[GP1:90,2] + 36.822;
   1:L PR[91] 10mm/sec CNT100;
   1:  PR[GP1:91,1] = PR[GP1:90,1] + 16.303;
   1:  PR[GP1:91,2] = PR[GP1:90,2] + 36.194;
   1:L PR[91] 10mm/sec CNT100;
   1:  PR[GP1:91,1] = PR[GP1:90,1] + 6.896;
   1:  PR[GP1:91,2] = PR[GP1:90,2] + 32.933;
   1:L PR[91] 10mm/sec CNT100;
   1:  PR[GP1:91,1] = PR[GP1:90,1] + 5.454;
   1:  PR[GP1:91,2] = PR[GP1:90,2] + 32.180;
   1:L PR[91] 10mm/sec CNT100;
   1:  PR[GP1:91,1] = PR[GP1:90,1] + 3.623;
   1:  PR[GP1:91,2] = PR[GP1:90,2] + 30.887;
   1:L PR[91] 10mm/sec CNT100;
   1:  PR[GP1:91,1] = PR[GP1:90,1] + 3.627;
   1:  PR[GP1:91,2] = PR[GP1:90,2] + 30.804;
   1:L PR[91] 10mm/sec CNT100;
   1:  PR[GP1:91,1] = PR[GP1:90,1] + 2.045;
   1:  PR[GP1:91,2] = PR[GP1:90,2] + 29.923;
   1:L PR[91] 10mm/sec CNT100;
   1:  PR[GP1:91,1] = PR[GP1:90,1] + -0.535;
   1:  PR[GP1:91,2] = PR[GP1:90,2] + 30.670;
   1:  PR[GP1:91,3] = PR[GP1:90,3] + 63.840;
   1:L PR[91] 10mm/sec CNT100;
   1:  PR[GP1:91,1] = PR[GP1:90,1] + -2.382;
   1:  PR[GP1:91,2] = PR[GP1:90,2] + 31.100;
   1:L PR[91] 10mm/sec CNT100;
   1:  PR[GP1:91,1] = PR[GP1:90,1] + -4.176;
   1:  PR[GP1:91,2] = PR[GP1:90,2] + 32.367;
   1:L PR[91] 10mm/sec CNT100;
   1:  PR[GP1:91,1] = PR[GP1:90,1] + -5.334;
   1:  PR[GP1:91,2] = PR[GP1:90,2] + 32.973;
   1:L PR[91] 10mm/sec CNT100;
   1:  PR[GP1:91,1] = PR[GP1:90,1] + -6.796;
   1:  PR[GP1:91,2] = PR[GP1:90,2] + 33.443;
   1:L PR[91] 10mm/sec CNT100;
   1:  PR[GP1:91,1] = PR[GP1:90,1] + -17.033;
   1:  PR[GP1:91,2] = PR[GP1:90,2] + 36.982;
   1:L PR[91] 10mm/sec CNT100;
   1:  PR[GP1:91,1] = PR[GP1:90,1] + -18.972;
   1:  PR[GP1:91,2] = PR[GP1:90,2] + 37.235;
   1:L PR[91] 10mm/sec CNT100;
   1:  PR[GP1:91,1] = PR[GP1:90,1] + -21.292;
   1:  PR[GP1:91,2] = PR[GP1:90,2] + 37.156;
   1:L PR[91] 10mm/sec CNT100;
   1:  PR[GP1:91,1] = PR[GP1:90,1] + -30.894;
   1:  PR[GP1:91,2] = PR[GP1:90,2] + 37.107;
   1:L PR[91] 10mm/sec CNT100;
   1:  PR[GP1:91,1] = PR[GP1:90,1] + -33.510;
   1:  PR[GP1:91,2] = PR[GP1:90,2] + 36.543;
   1:L PR[91] 10mm/sec CNT100;
   1:  PR[GP1:91,1] = PR[GP1:90,1] + -36.413;
   1:  PR[GP1:91,2] = PR[GP1:90,2] + 35.394;
   1:L PR[91] 10mm/sec CNT100;
   1:  PR[GP1:91,1] = PR[GP1:90,1] + -43.983;
   1:  PR[GP1:91,2] = PR[GP1:90,2] + 32.706;
   1:L PR[91] 10mm/sec CNT100;
   1:  PR[GP1:91,1] = PR[GP1:90,1] + -46.847;
   1:  PR[GP1:91,2] = PR[GP1:90,2] + 30.922;
   1:L PR[91] 10mm/sec CNT100;
   1:  PR[GP1:91,1] = PR[GP1:90,1] + -49.655;
   1:  PR[GP1:91,2] = PR[GP1:90,2] + 28.428;
   1:L PR[91] 10mm/sec CNT100;
   1:  PR[GP1:91,1] = PR[GP1:90,1] + -54.714;
   1:  PR[GP1:91,2] = PR[GP1:90,2] + 24.334;
   1:L PR[91] 10mm/sec CNT100;
   1:  PR[GP1:91,1] = PR[GP1:90,1] + -57.058;
   1:  PR[GP1:91,2] = PR[GP1:90,2] + 21.283;
   1:L PR[91] 10mm/sec CNT100;
   1:  PR[GP1:91,1] = PR[GP1:90,1] + -59.042;
   1:  PR[GP1:91,2] = PR[GP1:90,2] + 17.434;
   1:L PR[91] 10mm/sec CNT100;
   1:  PR[GP1:91,1] = PR[GP1:90,1] + -61.806;
   1:  PR[GP1:91,2] = PR[GP1:90,2] + 12.817;
   1:L PR[91] 10mm/sec CNT100;
   1:  PR[GP1:91,1] = PR[GP1:90,1] + -62.957;
   1:  PR[GP1:91,2] = PR[GP1:90,2] + 8.912;
   1:L PR[91] 10mm/sec CNT100;
   1:  PR[GP1:91,1] = PR[GP1:90,1] + -63.339;
   1:  PR[GP1:91,2] = PR[GP1:90,2] + 4.733;
   1:L PR[91] 10mm/sec CNT100;
   1:  PR[GP1:91,1] = PR[GP1:90,1] + -64.218;
   1:  PR[GP1:91,2] = PR[GP1:90,2] + -0.032;
   1:L PR[91] 10mm/sec CNT100;
   1:  PR[GP1:91,1] = PR[GP1:90,1] + -63.846;
   1:  PR[GP1:91,2] = PR[GP1:90,2] + -4.145;
   1:L PR[91] 10mm/sec CNT100;
   1:  PR[GP1:91,1] = PR[GP1:90,1] + -62.964;
   1:  PR[GP1:91,2] = PR[GP1:90,2] + -8.896;
   1:L PR[91] 10mm/sec CNT100;
   1:  PR[GP1:91,1] = PR[GP1:90,1] + -61.799;
   1:  PR[GP1:91,2] = PR[GP1:90,2] + -12.847;
   1:L PR[91] 10mm/sec CNT100;
   1:  PR[GP1:91,1] = PR[GP1:90,1] + -59.914;
   1:  PR[GP1:91,2] = PR[GP1:90,2] + -16.543;
   1:L PR[91] 10mm/sec CNT100;
   1:  PR[GP1:91,1] = PR[GP1:90,1] + -57.068;
   1:  PR[GP1:91,2] = PR[GP1:90,2] + -21.279;
   1:L PR[91] 10mm/sec CNT100;
   1:  PR[GP1:91,1] = PR[GP1:90,1] + -54.702;
   1:  PR[GP1:91,2] = PR[GP1:90,2] + -24.358;
   1:L PR[91] 10mm/sec CNT100;
   1:  PR[GP1:91,1] = PR[GP1:90,1] + -52.043;
   1:  PR[GP1:91,2] = PR[GP1:90,2] + -26.743;
   1:L PR[91] 10mm/sec CNT100;
   1:  PR[GP1:91,1] = PR[GP1:90,1] + -46.853;
   1:  PR[GP1:91,2] = PR[GP1:90,2] + -30.926;
   1:L PR[91] 10mm/sec CNT100;
   1:  PR[GP1:91,1] = PR[GP1:90,1] + -43.967;
   1:  PR[GP1:91,2] = PR[GP1:90,2] + -32.724;
   1:L PR[91] 10mm/sec CNT100;
   1:  PR[GP1:91,1] = PR[GP1:90,1] + -41.141;
   1:  PR[GP1:91,2] = PR[GP1:90,2] + -33.859;
   1:L PR[91] 10mm/sec CNT100;
   1:  PR[GP1:91,1] = PR[GP1:90,1] + -33.510;
   1:  PR[GP1:91,2] = PR[GP1:90,2] + -36.552;
   1:L PR[91] 10mm/sec CNT100;
   1:  PR[GP1:91,1] = PR[GP1:90,1] + -30.873;
   1:  PR[GP1:91,2] = PR[GP1:90,2] + -37.120;
   1:L PR[91] 10mm/sec CNT100;
   1:  PR[GP1:91,1] = PR[GP1:90,1] + -28.477;
   1:  PR[GP1:91,2] = PR[GP1:90,2] + -37.213;
   1:L PR[91] 10mm/sec CNT100;
   1:  PR[GP1:91,1] = PR[GP1:90,1] + -18.965;
   1:  PR[GP1:91,2] = PR[GP1:90,2] + -37.243;
   1:L PR[91] 10mm/sec CNT100;
   1:  PR[GP1:91,1] = PR[GP1:90,1] + -17.010;
   1:  PR[GP1:91,2] = PR[GP1:90,2] + -36.987;
   1:L PR[91] 10mm/sec CNT100;
   1:  PR[GP1:91,1] = PR[GP1:90,1] + -15.325;
   1:  PR[GP1:91,2] = PR[GP1:90,2] + -36.451;
   1:L PR[91] 10mm/sec CNT100;
   1:  PR[GP1:91,1] = PR[GP1:90,1] + -5.324;
   1:  PR[GP1:91,2] = PR[GP1:90,2] + -32.976;
   1:L PR[91] 10mm/sec CNT100;
   1:  PR[GP1:91,1] = PR[GP1:90,1] + -4.169;
   1:  PR[GP1:91,2] = PR[GP1:90,2] + -32.371;
   1:L PR[91] 10mm/sec CNT100;
   1:  PR[GP1:91,1] = PR[GP1:90,1] + -2.339;
   1:  PR[GP1:91,2] = PR[GP1:90,2] + -31.042;
   1:L PR[91] 10mm/sec CNT100;
   1:  PR[GP1:91,1] = PR[GP1:90,1] + -0.346;
   1:  PR[GP1:91,2] = PR[GP1:90,2] + -30.962;
   1:L PR[91] 10mm/sec CNT100;
   1:  PR[GP1:91,1] = PR[GP1:90,1] + 2.136;
   1:  PR[GP1:91,2] = PR[GP1:90,2] + -30.432;
   1:L PR[91] 10mm/sec CNT100;
   1:  PR[GP1:91,1] = PR[GP1:90,1] + 2.553;
   1:  PR[GP1:91,2] = PR[GP1:90,2] + -30.767;
   1:L PR[91] 10mm/sec CNT100;
   1:  PR[GP1:91,1] = PR[GP1:90,1] + 3.260;
   1:  PR[GP1:91,2] = PR[GP1:90,2] + -31.119;
   1:L PR[91] 10mm/sec CNT100;
   1:  PR[GP1:91,1] = PR[GP1:90,1] + 4.987;
   1:  PR[GP1:91,2] = PR[GP1:90,2] + -32.374;
   1:L PR[91] 10mm/sec CNT100;
   1:  PR[GP1:91,1] = PR[GP1:90,1] + 6.128;
   1:  PR[GP1:91,2] = PR[GP1:90,2] + -32.970;
   1:L PR[91] 10mm/sec CNT100;
   1:  PR[GP1:91,1] = PR[GP1:90,1] + 7.583;
   1:  PR[GP1:91,2] = PR[GP1:90,2] + -33.437;
   1:L PR[91] 10mm/sec CNT100;
   1:  PR[GP1:91,1] = PR[GP1:90,1] + 17.834;
   1:  PR[GP1:91,2] = PR[GP1:90,2] + -36.986;
   1:L PR[91] 10mm/sec CNT100;
   1:  PR[GP1:91,1] = PR[GP1:90,1] + 19.769;
   1:  PR[GP1:91,2] = PR[GP1:90,2] + -37.241;
   1:L PR[91] 10mm/sec CNT100;
   1:  PR[GP1:91,1] = PR[GP1:90,1] + 22.078;
   1:  PR[GP1:91,2] = PR[GP1:90,2] + -37.163;
   1:L PR[91] 10mm/sec CNT100;
   1:  PR[GP1:91,1] = PR[GP1:90,1] + 31.685;
   1:  PR[GP1:91,2] = PR[GP1:90,2] + -37.121;
   1:L PR[91] 10mm/sec CNT100;
   1:  PR[GP1:91,1] = PR[GP1:90,1] + 34.297;
   1:  PR[GP1:91,2] = PR[GP1:90,2] + -36.559;
   1:L PR[91] 10mm/sec CNT100;
   1:  PR[GP1:91,1] = PR[GP1:90,1] + 37.204;
   1:  PR[GP1:91,2] = PR[GP1:90,2] + -35.414;
   1:L PR[91] 10mm/sec CNT100;
   1:  PR[GP1:91,1] = PR[GP1:90,1] + 44.781;
   1:  PR[GP1:91,2] = PR[GP1:90,2] + -32.728;
   1:L PR[91] 10mm/sec CNT100;
   1:  PR[GP1:91,1] = PR[GP1:90,1] + 47.627;
   1:  PR[GP1:91,2] = PR[GP1:90,2] + -30.964;
   1:L PR[91] 10mm/sec CNT100;
   1:  PR[GP1:91,1] = PR[GP1:90,1] + 50.418;
   1:  PR[GP1:91,2] = PR[GP1:90,2] + -28.492;
   1:L PR[91] 10mm/sec CNT100;
   1:  PR[GP1:91,1] = PR[GP1:90,1] + 55.484;
   1:  PR[GP1:91,2] = PR[GP1:90,2] + -24.392;
   1:L PR[91] 10mm/sec CNT100;
   1:  PR[GP1:91,1] = PR[GP1:90,1] + 57.853;
   1:  PR[GP1:91,2] = PR[GP1:90,2] + -21.316;
   1:L PR[91] 10mm/sec CNT100;
   1:  PR[GP1:91,1] = PR[GP1:90,1] + 59.842;
   1:  PR[GP1:91,2] = PR[GP1:90,2] + -17.499;
   1:L PR[91] 10mm/sec CNT100;
   1:  PR[GP1:91,1] = PR[GP1:90,1] + 62.609;
   1:  PR[GP1:91,2] = PR[GP1:90,2] + -12.890;
   1:L PR[91] 10mm/sec CNT100;
   1:  PR[GP1:91,1] = PR[GP1:90,1] + 63.758;
   1:  PR[GP1:91,2] = PR[GP1:90,2] + -9.043;
   1:L PR[91] 10mm/sec CNT100;
   1:  PR[GP1:91,1] = PR[GP1:90,1] + 64.159;
   1:  PR[GP1:91,2] = PR[GP1:90,2] + -4.749;
   1:L PR[91] 10mm/sec CNT100;
   1:  PR[GP1:91,1] = PR[GP1:90,1] + 65.038;
   1:  PR[GP1:91,2] = PR[GP1:90,2] + 0.023;
   1:L PR[91] 10mm/sec CNT100;
   1:  PR[GP1:91,1] = PR[GP1:90,1] + 64.648;
   1:  PR[GP1:91,2] = PR[GP1:90,2] + 4.250;
   1:L PR[91] 10mm/sec CNT100;
   1:  PR[GP1:91,1] = PR[GP1:90,1] + 63.766;
   1:  PR[GP1:91,2] = PR[GP1:90,2] + 9.007;
   1:L PR[91] 10mm/sec CNT100;
   1:  PR[GP1:91,1] = PR[GP1:90,1] + 62.604;
   1:  PR[GP1:91,2] = PR[GP1:90,2] + 12.898;
   1:L PR[91] 10mm/sec CNT100;
   1:  PR[GP1:91,1] = PR[GP1:90,1] + 60.713;
   1:  PR[GP1:91,2] = PR[GP1:90,2] + 16.563;
   1:L PR[91] 10mm/sec CNT100;
   1:  PR[GP1:91,1] = PR[GP1:90,1] + 57.867;
   1:  PR[GP1:91,2] = PR[GP1:90,2] + 21.290;
   1:L PR[91] 10mm/sec CNT100;
   1:  PR[GP1:91,1] = PR[GP1:90,1] + 55.477;
   1:  PR[GP1:91,2] = PR[GP1:90,2] + 24.392;
   1:L PR[91] 10mm/sec CNT100;
   1:  PR[GP1:91,1] = PR[GP1:90,1] + 52.833;
   1:  PR[GP1:91,2] = PR[GP1:90,2] + 26.757;
   1:L PR[91] 10mm/sec CNT100;
   1:  PR[GP1:91,1] = PR[GP1:90,1] + 47.644;
   1:  PR[GP1:91,2] = PR[GP1:90,2] + 30.945;
   1:L PR[91] 10mm/sec CNT100;
   1:  PR[GP1:91,1] = PR[GP1:90,1] + 44.777;
   1:  PR[GP1:91,2] = PR[GP1:90,2] + 32.723;
   1:L PR[91] 10mm/sec CNT100;
   1:  PR[GP1:91,1] = PR[GP1:90,1] + 41.947;
   1:  PR[GP1:91,2] = PR[GP1:90,2] + 33.853;
   1:L PR[91] 10mm/sec CNT100;
   1:  PR[GP1:91,1] = PR[GP1:90,1] + 34.319;
   1:  PR[GP1:91,2] = PR[GP1:90,2] + 36.546;
   1:L PR[91] 10mm/sec CNT100;
   1:  PR[GP1:91,1] = PR[GP1:90,1] + 31.686;
   1:  PR[GP1:91,2] = PR[GP1:90,2] + 37.112;
   1:L PR[91] 10mm/sec CNT100;
   1:  PR[GP1:91,1] = PR[GP1:90,1] + 29.302;
   1:  PR[GP1:91,2] = PR[GP1:90,2] + 37.202;
   1:L PR[91] 10mm/sec CNT100;
   1:  PR[GP1:91,1] = PR[GP1:90,1] + 19.794;
   1:  PR[GP1:91,2] = PR[GP1:90,2] + 37.236;
   1:L PR[91] 10mm/sec CNT100;
   1:  PR[GP1:91,1] = PR[GP1:90,1] + 17.842;
   1:  PR[GP1:91,2] = PR[GP1:90,2] + 36.979;
   1:L PR[91] 10mm/sec CNT100;
   1:  PR[GP1:91,1] = PR[GP1:90,1] + 16.155;
   1:  PR[GP1:91,2] = PR[GP1:90,2] + 36.442;
   1:L PR[91] 10mm/sec CNT100;
   1:  PR[GP1:91,1] = PR[GP1:90,1] + 6.151;
   1:  PR[GP1:91,2] = PR[GP1:90,2] + 32.974;
   1:L PR[91] 10mm/sec CNT100;
   1:  PR[GP1:91,1] = PR[GP1:90,1] + 4.993;
   1:  PR[GP1:91,2] = PR[GP1:90,2] + 32.370;
   1:L PR[91] 10mm/sec CNT100;
   1:  PR[GP1:91,1] = PR[GP1:90,1] + 3.562;
   1:  PR[GP1:91,2] = PR[GP1:90,2] + 31.359;
   1:L PR[91] 10mm/sec CNT100;
   1:  PR[GP1:91,1] = PR[GP1:90,1] + 3.567;
   1:  PR[GP1:91,2] = PR[GP1:90,2] + 31.264;
   1:L PR[91] 10mm/sec CNT100;
   1:  PR[GP1:91,1] = PR[GP1:90,1] + 2.110;
   1:  PR[GP1:91,2] = PR[GP1:90,2] + 30.453;
   1:L PR[91] 10mm/sec CNT100;
   1:  PR[GP1:91,1] = PR[GP1:90,1] + -0.864;
   1:  PR[GP1:91,2] = PR[GP1:90,2] + 31.233;
   1:  PR[GP1:91,3] = PR[GP1:90,3] + 65.170;
   1:L PR[91] 10mm/sec CNT100;
   1:  PR[GP1:91,1] = PR[GP1:90,1] + -2.322;
   1:  PR[GP1:91,2] = PR[GP1:90,2] + 31.572;
   1:L PR[91] 10mm/sec CNT100;
   1:  PR[GP1:91,1] = PR[GP1:90,1] + -3.716;
   1:  PR[GP1:91,2] = PR[GP1:90,2] + 32.557;
   1:L PR[91] 10mm/sec CNT100;
   1:  PR[GP1:91,1] = PR[GP1:90,1] + -4.589;
   1:  PR[GP1:91,2] = PR[GP1:90,2] + 33.014;
   1:L PR[91] 10mm/sec CNT100;
   1:  PR[GP1:91,1] = PR[GP1:90,1] + -5.704;
   1:  PR[GP1:91,2] = PR[GP1:90,2] + 33.372;
   1:L PR[91] 10mm/sec CNT100;
   1:  PR[GP1:91,1] = PR[GP1:90,1] + -16.601;
   1:  PR[GP1:91,2] = PR[GP1:90,2] + 37.140;
   1:L PR[91] 10mm/sec CNT100;
   1:  PR[GP1:91,1] = PR[GP1:90,1] + -18.205;
   1:  PR[GP1:91,2] = PR[GP1:90,2] + 37.349;
   1:L PR[91] 10mm/sec CNT100;
   1:  PR[GP1:91,1] = PR[GP1:90,1] + -20.140;
   1:  PR[GP1:91,2] = PR[GP1:90,2] + 37.283;
   1:L PR[91] 10mm/sec CNT100;
   1:  PR[GP1:91,1] = PR[GP1:90,1] + -30.484;
   1:  PR[GP1:91,2] = PR[GP1:90,2] + 37.231;
   1:L PR[91] 10mm/sec CNT100;
   1:  PR[GP1:91,1] = PR[GP1:90,1] + -32.756;
   1:  PR[GP1:91,2] = PR[GP1:90,2] + 36.741;
   1:L PR[91] 10mm/sec CNT100;
   1:  PR[GP1:91,1] = PR[GP1:90,1] + -35.288;
   1:  PR[GP1:91,2] = PR[GP1:90,2] + 35.738;
   1:L PR[91] 10mm/sec CNT100;
   1:  PR[GP1:91,1] = PR[GP1:90,1] + -43.583;
   1:  PR[GP1:91,2] = PR[GP1:90,2] + 32.793;
   1:L PR[91] 10mm/sec CNT100;
   1:  PR[GP1:91,1] = PR[GP1:90,1] + -46.139;
   1:  PR[GP1:91,2] = PR[GP1:90,2] + 31.201;
   1:L PR[91] 10mm/sec CNT100;
   1:  PR[GP1:91,1] = PR[GP1:90,1] + -48.651;
   1:  PR[GP1:91,2] = PR[GP1:90,2] + 28.970;
   1:L PR[91] 10mm/sec CNT100;
   1:  PR[GP1:91,1] = PR[GP1:90,1] + -54.314;
   1:  PR[GP1:91,2] = PR[GP1:90,2] + 24.387;
   1:L PR[91] 10mm/sec CNT100;
   1:  PR[GP1:91,1] = PR[GP1:90,1] + -56.438;
   1:  PR[GP1:91,2] = PR[GP1:90,2] + 21.623;
   1:L PR[91] 10mm/sec CNT100;
   1:  PR[GP1:91,1] = PR[GP1:90,1] + -58.239;
   1:  PR[GP1:91,2] = PR[GP1:90,2] + 18.128;
   1:L PR[91] 10mm/sec CNT100;
   1:  PR[GP1:91,1] = PR[GP1:90,1] + -61.398;
   1:  PR[GP1:91,2] = PR[GP1:90,2] + 12.851;
   1:L PR[91] 10mm/sec CNT100;
   1:  PR[GP1:91,1] = PR[GP1:90,1] + -62.449;
   1:  PR[GP1:91,2] = PR[GP1:90,2] + 9.286;
   1:L PR[91] 10mm/sec CNT100;
   1:  PR[GP1:91,1] = PR[GP1:90,1] + -62.799;
   1:  PR[GP1:91,2] = PR[GP1:90,2] + 5.462;
   1:L PR[91] 10mm/sec CNT100;
   1:  PR[GP1:91,1] = PR[GP1:90,1] + -63.811;
   1:  PR[GP1:91,2] = PR[GP1:90,2] + -0.032;
   1:L PR[91] 10mm/sec CNT100;
   1:  PR[GP1:91,1] = PR[GP1:90,1] + -63.471;
   1:  PR[GP1:91,2] = PR[GP1:90,2] + -3.803;
   1:L PR[91] 10mm/sec CNT100;
   1:  PR[GP1:91,1] = PR[GP1:90,1] + -62.456;
   1:  PR[GP1:91,2] = PR[GP1:90,2] + -9.270;
   1:L PR[91] 10mm/sec CNT100;
   1:  PR[GP1:91,1] = PR[GP1:90,1] + -61.391;
   1:  PR[GP1:91,2] = PR[GP1:90,2] + -12.882;
   1:L PR[91] 10mm/sec CNT100;
   1:  PR[GP1:91,1] = PR[GP1:90,1] + -59.668;
   1:  PR[GP1:91,2] = PR[GP1:90,2] + -16.260;
   1:L PR[91] 10mm/sec CNT100;
   1:  PR[GP1:91,1] = PR[GP1:90,1] + -56.447;
   1:  PR[GP1:91,2] = PR[GP1:90,2] + -21.619;
   1:L PR[91] 10mm/sec CNT100;
   1:  PR[GP1:91,1] = PR[GP1:90,1] + -54.302;
   1:  PR[GP1:91,2] = PR[GP1:90,2] + -24.411;
   1:L PR[91] 10mm/sec CNT100;
   1:  PR[GP1:91,1] = PR[GP1:90,1] + -51.891;
   1:  PR[GP1:91,2] = PR[GP1:90,2] + -26.574;
   1:L PR[91] 10mm/sec CNT100;
   1:  PR[GP1:91,1] = PR[GP1:90,1] + -46.144;
   1:  PR[GP1:91,2] = PR[GP1:90,2] + -31.206;
   1:L PR[91] 10mm/sec CNT100;
   1:  PR[GP1:91,1] = PR[GP1:90,1] + -43.566;
   1:  PR[GP1:91,2] = PR[GP1:90,2] + -32.812;
   1:L PR[91] 10mm/sec CNT100;
   1:  PR[GP1:91,1] = PR[GP1:90,1] + -41.041;
   1:  PR[GP1:91,2] = PR[GP1:90,2] + -33.826;
   1:L PR[91] 10mm/sec CNT100;
   1:  PR[GP1:91,1] = PR[GP1:90,1] + -32.755;
   1:  PR[GP1:91,2] = PR[GP1:90,2] + -36.749;
   1:L PR[91] 10mm/sec CNT100;
   1:  PR[GP1:91,1] = PR[GP1:90,1] + -30.462;
   1:  PR[GP1:91,2] = PR[GP1:90,2] + -37.244;
   1:L PR[91] 10mm/sec CNT100;
   1:  PR[GP1:91,1] = PR[GP1:90,1] + -28.377;
   1:  PR[GP1:91,2] = PR[GP1:90,2] + -37.324;
   1:L PR[91] 10mm/sec CNT100;
   1:  PR[GP1:91,1] = PR[GP1:90,1] + -18.197;
   1:  PR[GP1:91,2] = PR[GP1:90,2] + -37.356;
   1:L PR[91] 10mm/sec CNT100;
   1:  PR[GP1:91,1] = PR[GP1:90,1] + -16.576;
   1:  PR[GP1:91,2] = PR[GP1:90,2] + -37.145;
   1:L PR[91] 10mm/sec CNT100;
   1:  PR[GP1:91,1] = PR[GP1:90,1] + -15.176;
   1:  PR[GP1:91,2] = PR[GP1:90,2] + -36.699;
   1:L PR[91] 10mm/sec CNT100;
   1:  PR[GP1:91,1] = PR[GP1:90,1] + -4.578;
   1:  PR[GP1:91,2] = PR[GP1:90,2] + -33.016;
   1:L PR[91] 10mm/sec CNT100;
   1:  PR[GP1:91,1] = PR[GP1:90,1] + -3.709;
   1:  PR[GP1:91,2] = PR[GP1:90,2] + -32.562;
   1:L PR[91] 10mm/sec CNT100;
   1:  PR[GP1:91,1] = PR[GP1:90,1] + -2.278;
   1:  PR[GP1:91,2] = PR[GP1:90,2] + -31.522;
   1:L PR[91] 10mm/sec CNT100;
   1:  PR[GP1:91,1] = PR[GP1:90,1] + 0.015;
   1:  PR[GP1:91,2] = PR[GP1:90,2] + -31.430;
   1:L PR[91] 10mm/sec CNT100;
   1:  PR[GP1:91,1] = PR[GP1:90,1] + 2.203;
   1:  PR[GP1:91,2] = PR[GP1:90,2] + -30.963;
   1:L PR[91] 10mm/sec CNT100;
   1:  PR[GP1:91,1] = PR[GP1:90,1] + 2.659;
   1:  PR[GP1:91,2] = PR[GP1:90,2] + -31.330;
   1:L PR[91] 10mm/sec CNT100;
   1:  PR[GP1:91,1] = PR[GP1:90,1] + 3.198;
   1:  PR[GP1:91,2] = PR[GP1:90,2] + -31.599;
   1:L PR[91] 10mm/sec CNT100;
   1:  PR[GP1:91,1] = PR[GP1:90,1] + 4.526;
   1:  PR[GP1:91,2] = PR[GP1:90,2] + -32.564;
   1:L PR[91] 10mm/sec CNT100;
   1:  PR[GP1:91,1] = PR[GP1:90,1] + 5.382;
   1:  PR[GP1:91,2] = PR[GP1:90,2] + -33.010;
   1:L PR[91] 10mm/sec CNT100;
   1:  PR[GP1:91,1] = PR[GP1:90,1] + 6.490;
   1:  PR[GP1:91,2] = PR[GP1:90,2] + -33.366;
   1:L PR[91] 10mm/sec CNT100;
   1:  PR[GP1:91,1] = PR[GP1:90,1] + 17.401;
   1:  PR[GP1:91,2] = PR[GP1:90,2] + -37.144;
   1:L PR[91] 10mm/sec CNT100;
   1:  PR[GP1:91,1] = PR[GP1:90,1] + 19.002;
   1:  PR[GP1:91,2] = PR[GP1:90,2] + -37.354;
   1:L PR[91] 10mm/sec CNT100;
   1:  PR[GP1:91,1] = PR[GP1:90,1] + 20.927;
   1:  PR[GP1:91,2] = PR[GP1:90,2] + -37.290;
   1:L PR[91] 10mm/sec CNT100;
   1:  PR[GP1:91,1] = PR[GP1:90,1] + 31.277;
   1:  PR[GP1:91,2] = PR[GP1:90,2] + -37.244;
   1:L PR[91] 10mm/sec CNT100;
   1:  PR[GP1:91,1] = PR[GP1:90,1] + 33.545;
   1:  PR[GP1:91,2] = PR[GP1:90,2] + -36.756;
   1:L PR[91] 10mm/sec CNT100;
   1:  PR[GP1:91,1] = PR[GP1:90,1] + 36.080;
   1:  PR[GP1:91,2] = PR[GP1:90,2] + -35.757;
   1:L PR[91] 10mm/sec CNT100;
   1:  PR[GP1:91,1] = PR[GP1:90,1] + 44.382;
   1:  PR[GP1:91,2] = PR[GP1:90,2] + -32.815;
   1:L PR[91] 10mm/sec CNT100;
   1:  PR[GP1:91,1] = PR[GP1:90,1] + 46.921;
   1:  PR[GP1:91,2] = PR[GP1:90,2] + -31.241;
   1:L PR[91] 10mm/sec CNT100;
   1:  PR[GP1:91,1] = PR[GP1:90,1] + 49.419;
   1:  PR[GP1:91,2] = PR[GP1:90,2] + -29.029;
   1:L PR[91] 10mm/sec CNT100;
   1:  PR[GP1:91,1] = PR[GP1:90,1] + 55.088;
   1:  PR[GP1:91,2] = PR[GP1:90,2] + -24.440;
   1:L PR[91] 10mm/sec CNT100;
   1:  PR[GP1:91,1] = PR[GP1:90,1] + 57.234;
   1:  PR[GP1:91,2] = PR[GP1:90,2] + -21.654;
   1:L PR[91] 10mm/sec CNT100;
   1:  PR[GP1:91,1] = PR[GP1:90,1] + 59.041;
   1:  PR[GP1:91,2] = PR[GP1:90,2] + -18.188;
   1:L PR[91] 10mm/sec CNT100;
   1:  PR[GP1:91,1] = PR[GP1:90,1] + 62.202;
   1:  PR[GP1:91,2] = PR[GP1:90,2] + -12.921;
   1:L PR[91] 10mm/sec CNT100;
   1:  PR[GP1:91,1] = PR[GP1:90,1] + 63.251;
   1:  PR[GP1:91,2] = PR[GP1:90,2] + -9.409;
   1:L PR[91] 10mm/sec CNT100;
   1:  PR[GP1:91,1] = PR[GP1:90,1] + 63.619;
   1:  PR[GP1:91,2] = PR[GP1:90,2] + -5.480;
   1:L PR[91] 10mm/sec CNT100;
   1:  PR[GP1:91,1] = PR[GP1:90,1] + 64.632;
   1:  PR[GP1:91,2] = PR[GP1:90,2] + 0.023;
   1:L PR[91] 10mm/sec CNT100;
   1:  PR[GP1:91,1] = PR[GP1:90,1] + 64.274;
   1:  PR[GP1:91,2] = PR[GP1:90,2] + 3.900;
   1:L PR[91] 10mm/sec CNT100;
   1:  PR[GP1:91,1] = PR[GP1:90,1] + 63.260;
   1:  PR[GP1:91,2] = PR[GP1:90,2] + 9.372;
   1:L PR[91] 10mm/sec CNT100;
   1:  PR[GP1:91,1] = PR[GP1:90,1] + 62.197;
   1:  PR[GP1:91,2] = PR[GP1:90,2] + 12.929;
   1:L PR[91] 10mm/sec CNT100;
   1:  PR[GP1:91,1] = PR[GP1:90,1] + 60.469;
   1:  PR[GP1:91,2] = PR[GP1:90,2] + 16.278;
   1:L PR[91] 10mm/sec CNT100;
   1:  PR[GP1:91,1] = PR[GP1:90,1] + 57.248;
   1:  PR[GP1:91,2] = PR[GP1:90,2] + 21.628;
   1:L PR[91] 10mm/sec CNT100;
   1:  PR[GP1:91,1] = PR[GP1:90,1] + 55.082;
   1:  PR[GP1:91,2] = PR[GP1:90,2] + 24.440;
   1:L PR[91] 10mm/sec CNT100;
   1:  PR[GP1:91,1] = PR[GP1:90,1] + 52.683;
   1:  PR[GP1:91,2] = PR[GP1:90,2] + 26.585;
   1:L PR[91] 10mm/sec CNT100;
   1:  PR[GP1:91,1] = PR[GP1:90,1] + 46.939;
   1:  PR[GP1:91,2] = PR[GP1:90,2] + 31.222;
   1:L PR[91] 10mm/sec CNT100;
   1:  PR[GP1:91,1] = PR[GP1:90,1] + 44.378;
   1:  PR[GP1:91,2] = PR[GP1:90,2] + 32.809;
   1:L PR[91] 10mm/sec CNT100;
   1:  PR[GP1:91,1] = PR[GP1:90,1] + 41.850;
   1:  PR[GP1:91,2] = PR[GP1:90,2] + 33.819;
   1:L PR[91] 10mm/sec CNT100;
   1:  PR[GP1:91,1] = PR[GP1:90,1] + 33.567;
   1:  PR[GP1:91,2] = PR[GP1:90,2] + 36.743;
   1:L PR[91] 10mm/sec CNT100;
   1:  PR[GP1:91,1] = PR[GP1:90,1] + 31.279;
   1:  PR[GP1:91,2] = PR[GP1:90,2] + 37.236;
   1:L PR[91] 10mm/sec CNT100;
   1:  PR[GP1:91,1] = PR[GP1:90,1] + 29.203;
   1:  PR[GP1:91,2] = PR[GP1:90,2] + 37.314;
   1:L PR[91] 10mm/sec CNT100;
   1:  PR[GP1:91,1] = PR[GP1:90,1] + 19.028;
   1:  PR[GP1:91,2] = PR[GP1:90,2] + 37.350;
   1:L PR[91] 10mm/sec CNT100;
   1:  PR[GP1:91,1] = PR[GP1:90,1] + 17.410;
   1:  PR[GP1:91,2] = PR[GP1:90,2] + 37.137;
   1:L PR[91] 10mm/sec CNT100;
   1:  PR[GP1:91,1] = PR[GP1:90,1] + 16.007;
   1:  PR[GP1:91,2] = PR[GP1:90,2] + 36.691;
   1:L PR[91] 10mm/sec CNT100;
   1:  PR[GP1:91,1] = PR[GP1:90,1] + 5.406;
   1:  PR[GP1:91,2] = PR[GP1:90,2] + 33.015;
   1:L PR[91] 10mm/sec CNT100;
   1:  PR[GP1:91,1] = PR[GP1:90,1] + 4.533;
   1:  PR[GP1:91,2] = PR[GP1:90,2] + 32.559;
   1:L PR[91] 10mm/sec CNT100;
   1:  PR[GP1:91,1] = PR[GP1:90,1] + 3.501;
   1:  PR[GP1:91,2] = PR[GP1:90,2] + 31.831;
   1:L PR[91] 10mm/sec CNT100;
   1:  PR[GP1:91,1] = PR[GP1:90,1] + 3.507;
   1:  PR[GP1:91,2] = PR[GP1:90,2] + 31.724;
   1:L PR[91] 10mm/sec CNT100;
   1:  PR[GP1:91,1] = PR[GP1:90,1] + 2.176;
   1:  PR[GP1:91,2] = PR[GP1:90,2] + 30.984;
   1:L PR[91] 10mm/sec CNT100;
   1:  PR[GP1:91,1] = PR[GP1:90,1] + -1.193;
   1:  PR[GP1:91,2] = PR[GP1:90,2] + 31.796;
   1:  PR[GP1:91,3] = PR[GP1:90,3] + 66.500;
   1:L PR[91] 10mm/sec CNT100;
   1:  PR[GP1:91,1] = PR[GP1:90,1] + -2.261;
   1:  PR[GP1:91,2] = PR[GP1:90,2] + 32.044;
   1:L PR[91] 10mm/sec CNT100;
   1:  PR[GP1:91,1] = PR[GP1:90,1] + -3.257;
   1:  PR[GP1:91,2] = PR[GP1:90,2] + 32.748;
   1:L PR[91] 10mm/sec CNT100;
   1:  PR[GP1:91,1] = PR[GP1:90,1] + -3.844;
   1:  PR[GP1:91,2] = PR[GP1:90,2] + 33.055;
   1:L PR[91] 10mm/sec CNT100;
   1:  PR[GP1:91,1] = PR[GP1:90,1] + -4.612;
   1:  PR[GP1:91,2] = PR[GP1:90,2] + 33.302;
   1:L PR[91] 10mm/sec CNT100;
   1:  PR[GP1:91,1] = PR[GP1:90,1] + -16.168;
   1:  PR[GP1:91,2] = PR[GP1:90,2] + 37.297;
   1:L PR[91] 10mm/sec CNT100;
   1:  PR[GP1:91,1] = PR[GP1:90,1] + -17.439;
   1:  PR[GP1:91,2] = PR[GP1:90,2] + 37.463;
   1:L PR[91] 10mm/sec CNT100;
   1:  PR[GP1:91,1] = PR[GP1:90,1] + -18.989;
   1:  PR[GP1:91,2] = PR[GP1:90,2] + 37.410;
   1:L PR[91] 10mm/sec CNT100;
   1:  PR[GP1:91,1] = PR[GP1:90,1] + -30.075;
   1:  PR[GP1:91,2] = PR[GP1:90,2] + 37.354;
   1:L PR[91] 10mm/sec CNT100;
   1:  PR[GP1:91,1] = PR[GP1:90,1] + -32.002;
   1:  PR[GP1:91,2] = PR[GP1:90,2] + 36.938;
   1:L PR[91] 10mm/sec CNT100;
   1:  PR[GP1:91,1] = PR[GP1:90,1] + -34.164;
   1:  PR[GP1:91,2] = PR[GP1:90,2] + 36.083;
   1:L PR[91] 10mm/sec CNT100;
   1:  PR[GP1:91,1] = PR[GP1:90,1] + -43.183;
   1:  PR[GP1:91,2] = PR[GP1:90,2] + 32.880;
   1:L PR[91] 10mm/sec CNT100;
   1:  PR[GP1:91,1] = PR[GP1:90,1] + -45.430;
   1:  PR[GP1:91,2] = PR[GP1:90,2] + 31.480;
   1:L PR[91] 10mm/sec CNT100;
   1:  PR[GP1:91,1] = PR[GP1:90,1] + -47.647;
   1:  PR[GP1:91,2] = PR[GP1:90,2] + 29.512;
   1:L PR[91] 10mm/sec CNT100;
   1:  PR[GP1:91,1] = PR[GP1:90,1] + -53.914;
   1:  PR[GP1:91,2] = PR[GP1:90,2] + 24.440;
   1:L PR[91] 10mm/sec CNT100;
   1:  PR[GP1:91,1] = PR[GP1:90,1] + -55.817;
   1:  PR[GP1:91,2] = PR[GP1:90,2] + 21.963;
   1:L PR[91] 10mm/sec CNT100;
   1:  PR[GP1:91,1] = PR[GP1:90,1] + -57.436;
   1:  PR[GP1:91,2] = PR[GP1:90,2] + 18.822;
   1:L PR[91] 10mm/sec CNT100;
   1:  PR[GP1:91,1] = PR[GP1:90,1] + -60.990;
   1:  PR[GP1:91,2] = PR[GP1:90,2] + 12.885;
   1:L PR[91] 10mm/sec CNT100;
   1:  PR[GP1:91,1] = PR[GP1:90,1] + -61.941;
   1:  PR[GP1:91,2] = PR[GP1:90,2] + 9.660;
   1:L PR[91] 10mm/sec CNT100;
   1:  PR[GP1:91,1] = PR[GP1:90,1] + -62.258;
   1:  PR[GP1:91,2] = PR[GP1:90,2] + 6.191;
   1:L PR[91] 10mm/sec CNT100;
   1:  PR[GP1:91,1] = PR[GP1:90,1] + -63.405;
   1:  PR[GP1:91,2] = PR[GP1:90,2] + -0.032;
   1:L PR[91] 10mm/sec CNT100;
   1:  PR[GP1:91,1] = PR[GP1:90,1] + -63.095;
   1:  PR[GP1:91,2] = PR[GP1:90,2] + -3.462;
   1:L PR[91] 10mm/sec CNT100;
   1:  PR[GP1:91,1] = PR[GP1:90,1] + -61.948;
   1:  PR[GP1:91,2] = PR[GP1:90,2] + -9.644;
   1:L PR[91] 10mm/sec CNT100;
   1:  PR[GP1:91,1] = PR[GP1:90,1] + -60.983;
   1:  PR[GP1:91,2] = PR[GP1:90,2] + -12.916;
   1:L PR[91] 10mm/sec CNT100;
   1:  PR[GP1:91,1] = PR[GP1:90,1] + -59.422;
   1:  PR[GP1:91,2] = PR[GP1:90,2] + -15.977;
   1:L PR[91] 10mm/sec CNT100;
   1:  PR[GP1:91,1] = PR[GP1:90,1] + -55.826;
   1:  PR[GP1:91,2] = PR[GP1:90,2] + -21.960;
   1:L PR[91] 10mm/sec CNT100;
   1:  PR[GP1:91,1] = PR[GP1:90,1] + -53.902;
   1:  PR[GP1:91,2] = PR[GP1:90,2] + -24.464;
   1:L PR[91] 10mm/sec CNT100;
   1:  PR[GP1:91,1] = PR[GP1:90,1] + -51.737;
   1:  PR[GP1:91,2] = PR[GP1:90,2] + -26.406;
   1:L PR[91] 10mm/sec CNT100;
   1:  PR[GP1:91,1] = PR[GP1:90,1] + -45.435;
   1:  PR[GP1:91,2] = PR[GP1:90,2] + -31.486;
   1:L PR[91] 10mm/sec CNT100;
   1:  PR[GP1:91,1] = PR[GP1:90,1] + -43.166;
   1:  PR[GP1:91,2] = PR[GP1:90,2] + -32.899;
   1:L PR[91] 10mm/sec CNT100;
   1:  PR[GP1:91,1] = PR[GP1:90,1] + -40.941;
   1:  PR[GP1:91,2] = PR[GP1:90,2] + -33.793;
   1:L PR[91] 10mm/sec CNT100;
   1:  PR[GP1:91,1] = PR[GP1:90,1] + -32.001;
   1:  PR[GP1:91,2] = PR[GP1:90,2] + -36.947;
   1:L PR[91] 10mm/sec CNT100;
   1:  PR[GP1:91,1] = PR[GP1:90,1] + -30.052;
   1:  PR[GP1:91,2] = PR[GP1:90,2] + -37.367;
   1:L PR[91] 10mm/sec CNT100;
   1:  PR[GP1:91,1] = PR[GP1:90,1] + -28.277;
   1:  PR[GP1:91,2] = PR[GP1:90,2] + -37.436;
   1:L PR[91] 10mm/sec CNT100;
   1:  PR[GP1:91,1] = PR[GP1:90,1] + -17.429;
   1:  PR[GP1:91,2] = PR[GP1:90,2] + -37.470;
   1:L PR[91] 10mm/sec CNT100;
   1:  PR[GP1:91,1] = PR[GP1:90,1] + -16.143;
   1:  PR[GP1:91,2] = PR[GP1:90,2] + -37.302;
   1:L PR[91] 10mm/sec CNT100;
   1:  PR[GP1:91,1] = PR[GP1:90,1] + -15.027;
   1:  PR[GP1:91,2] = PR[GP1:90,2] + -36.947;
   1:L PR[91] 10mm/sec CNT100;
   1:  PR[GP1:91,1] = PR[GP1:90,1] + -3.832;
   1:  PR[GP1:91,2] = PR[GP1:90,2] + -33.056;
   1:L PR[91] 10mm/sec CNT100;
   1:  PR[GP1:91,1] = PR[GP1:90,1] + -3.249;
   1:  PR[GP1:91,2] = PR[GP1:90,2] + -32.752;
   1:L PR[91] 10mm/sec CNT100;
   1:  PR[GP1:91,1] = PR[GP1:90,1] + -2.217;
   1:  PR[GP1:91,2] = PR[GP1:90,2] + -32.002;
   1:L PR[91] 10mm/sec CNT100;
   1:  PR[GP1:91,1] = PR[GP1:90,1] + 0.377;
   1:  PR[GP1:91,2] = PR[GP1:90,2] + -31.898;
   1:L PR[91] 10mm/sec CNT100;
   1:  PR[GP1:91,1] = PR[GP1:90,1] + 2.269;
   1:  PR[GP1:91,2] = PR[GP1:90,2] + -31.494;
   1:L PR[91] 10mm/sec CNT100;
   1:  PR[GP1:91,1] = PR[GP1:90,1] + 2.765;
   1:  PR[GP1:91,2] = PR[GP1:90,2] + -31.893;
   1:L PR[91] 10mm/sec CNT100;
   1:  PR[GP1:91,1] = PR[GP1:90,1] + 3.137;
   1:  PR[GP1:91,2] = PR[GP1:90,2] + -32.079;
   1:L PR[91] 10mm/sec CNT100;
   1:  PR[GP1:91,1] = PR[GP1:90,1] + 4.065;
   1:  PR[GP1:91,2] = PR[GP1:90,2] + -32.753;
   1:L PR[91] 10mm/sec CNT100;
   1:  PR[GP1:91,1] = PR[GP1:90,1] + 4.636;
   1:  PR[GP1:91,2] = PR[GP1:90,2] + -33.051;
   1:L PR[91] 10mm/sec CNT100;
   1:  PR[GP1:91,1] = PR[GP1:90,1] + 5.396;
   1:  PR[GP1:91,2] = PR[GP1:90,2] + -33.295;
   1:L PR[91] 10mm/sec CNT100;
   1:  PR[GP1:91,1] = PR[GP1:90,1] + 16.967;
   1:  PR[GP1:91,2] = PR[GP1:90,2] + -37.301;
   1:L PR[91] 10mm/sec CNT100;
   1:  PR[GP1:91,1] = PR[GP1:90,1] + 18.235;
   1:  PR[GP1:91,2] = PR[GP1:90,2] + -37.468;
   1:L PR[91] 10mm/sec CNT100;
   1:  PR[GP1:91,1] = PR[GP1:90,1] + 19.777;
   1:  PR[GP1:91,2] = PR[GP1:90,2] + -37.416;
   1:L PR[91] 10mm/sec CNT100;
   1:  PR[GP1:91,1] = PR[GP1:90,1] + 30.869;
   1:  PR[GP1:91,2] = PR[GP1:90,2] + -37.368;
   1:L PR[91] 10mm/sec CNT100;
   1:  PR[GP1:91,1] = PR[GP1:90,1] + 32.793;
   1:  PR[GP1:91,2] = PR[GP1:90,2] + -36.953;
   1:L PR[91] 10mm/sec CNT100;
   1:  PR[GP1:91,1] = PR[GP1:90,1] + 34.957;
   1:  PR[GP1:91,2] = PR[GP1:90,2] + -36.101;
   1:L PR[91] 10mm/sec CNT100;
   1:  PR[GP1:91,1] = PR[GP1:90,1] + 43.983;
   1:  PR[GP1:91,2] = PR[GP1:90,2] + -32.902;
   1:L PR[91] 10mm/sec CNT100;
   1:  PR[GP1:91,1] = PR[GP1:90,1] + 46.215;
   1:  PR[GP1:91,2] = PR[GP1:90,2] + -31.518;
   1:L PR[91] 10mm/sec CNT100;
   1:  PR[GP1:91,1] = PR[GP1:90,1] + 48.420;
   1:  PR[GP1:91,2] = PR[GP1:90,2] + -29.566;
   1:L PR[91] 10mm/sec CNT100;
   1:  PR[GP1:91,1] = PR[GP1:90,1] + 54.692;
   1:  PR[GP1:91,2] = PR[GP1:90,2] + -24.489;
   1:L PR[91] 10mm/sec CNT100;
   1:  PR[GP1:91,1] = PR[GP1:90,1] + 56.616;
   1:  PR[GP1:91,2] = PR[GP1:90,2] + -21.992;
   1:L PR[91] 10mm/sec CNT100;
   1:  PR[GP1:91,1] = PR[GP1:90,1] + 58.239;
   1:  PR[GP1:91,2] = PR[GP1:90,2] + -18.876;
   1:L PR[91] 10mm/sec CNT100;
   1:  PR[GP1:91,1] = PR[GP1:90,1] + 61.796;
   1:  PR[GP1:91,2] = PR[GP1:90,2] + -12.951;
   1:L PR[91] 10mm/sec CNT100;
   1:  PR[GP1:91,1] = PR[GP1:90,1] + 62.745;
   1:  PR[GP1:91,2] = PR[GP1:90,2] + -9.774;
   1:L PR[91] 10mm/sec CNT100;
   1:  PR[GP1:91,1] = PR[GP1:90,1] + 63.078;
   1:  PR[GP1:91,2] = PR[GP1:90,2] + -6.210;
   1:L PR[91] 10mm/sec CNT100;
   1:  PR[GP1:91,1] = PR[GP1:90,1] + 64.226;
   1:  PR[GP1:91,2] = PR[GP1:90,2] + 0.023;
   1:L PR[91] 10mm/sec CNT100;
   1:  PR[GP1:91,1] = PR[GP1:90,1] + 63.900;
   1:  PR[GP1:91,2] = PR[GP1:90,2] + 3.550;
   1:L PR[91] 10mm/sec CNT100;
   1:  PR[GP1:91,1] = PR[GP1:90,1] + 62.753;
   1:  PR[GP1:91,2] = PR[GP1:90,2] + 9.738;
   1:L PR[91] 10mm/sec CNT100;
   1:  PR[GP1:91,1] = PR[GP1:90,1] + 61.791;
   1:  PR[GP1:91,2] = PR[GP1:90,2] + 12.959;
   1:L PR[91] 10mm/sec CNT100;
   1:  PR[GP1:91,1] = PR[GP1:90,1] + 60.225;
   1:  PR[GP1:91,2] = PR[GP1:90,2] + 15.994;
   1:L PR[91] 10mm/sec CNT100;
   1:  PR[GP1:91,1] = PR[GP1:90,1] + 56.630;
   1:  PR[GP1:91,2] = PR[GP1:90,2] + 21.965;
   1:L PR[91] 10mm/sec CNT100;
   1:  PR[GP1:91,1] = PR[GP1:90,1] + 54.686;
   1:  PR[GP1:91,2] = PR[GP1:90,2] + 24.488;
   1:L PR[91] 10mm/sec CNT100;
   1:  PR[GP1:91,1] = PR[GP1:90,1] + 52.533;
   1:  PR[GP1:91,2] = PR[GP1:90,2] + 26.413;
   1:L PR[91] 10mm/sec CNT100;
   1:  PR[GP1:91,1] = PR[GP1:90,1] + 46.234;
   1:  PR[GP1:91,2] = PR[GP1:90,2] + 31.498;
   1:L PR[91] 10mm/sec CNT100;
   1:  PR[GP1:91,1] = PR[GP1:90,1] + 43.980;
   1:  PR[GP1:91,2] = PR[GP1:90,2] + 32.895;
   1:L PR[91] 10mm/sec CNT100;
   1:  PR[GP1:91,1] = PR[GP1:90,1] + 41.752;
   1:  PR[GP1:91,2] = PR[GP1:90,2] + 33.785;
   1:L PR[91] 10mm/sec CNT100;
   1:  PR[GP1:91,1] = PR[GP1:90,1] + 32.816;
   1:  PR[GP1:91,2] = PR[GP1:90,2] + 36.940;
   1:L PR[91] 10mm/sec CNT100;
   1:  PR[GP1:91,1] = PR[GP1:90,1] + 30.871;
   1:  PR[GP1:91,2] = PR[GP1:90,2] + 37.359;
   1:L PR[91] 10mm/sec CNT100;
   1:  PR[GP1:91,1] = PR[GP1:90,1] + 29.105;
   1:  PR[GP1:91,2] = PR[GP1:90,2] + 37.425;
   1:L PR[91] 10mm/sec CNT100;
   1:  PR[GP1:91,1] = PR[GP1:90,1] + 18.262;
   1:  PR[GP1:91,2] = PR[GP1:90,2] + 37.463;
   1:L PR[91] 10mm/sec CNT100;
   1:  PR[GP1:91,1] = PR[GP1:90,1] + 16.977;
   1:  PR[GP1:91,2] = PR[GP1:90,2] + 37.294;
   1:L PR[91] 10mm/sec CNT100;
   1:  PR[GP1:91,1] = PR[GP1:90,1] + 15.860;
   1:  PR[GP1:91,2] = PR[GP1:90,2] + 36.939;
   1:L PR[91] 10mm/sec CNT100;
   1:  PR[GP1:91,1] = PR[GP1:90,1] + 4.661;
   1:  PR[GP1:91,2] = PR[GP1:90,2] + 33.056;
   1:L PR[91] 10mm/sec CNT100;
   1:  PR[GP1:91,1] = PR[GP1:90,1] + 4.072;
   1:  PR[GP1:91,2] = PR[GP1:90,2] + 32.749;
   1:L PR[91] 10mm/sec CNT100;
   1:  PR[GP1:91,1] = PR[GP1:90,1] + 3.440;
   1:  PR[GP1:91,2] = PR[GP1:90,2] + 32.303;
   1:L PR[91] 10mm/sec CNT100;
   1:  PR[GP1:91,1] = PR[GP1:90,1] + 3.446;
   1:  PR[GP1:91,2] = PR[GP1:90,2] + 32.185;
   1:L PR[91] 10mm/sec CNT100;
   1:  PR[GP1:91,1] = PR[GP1:90,1] + 2.241;
   1:  PR[GP1:91,2] = PR[GP1:90,2] + 31.514;
   1:L PR[91] 10mm/sec CNT100;
   1:  PR[GP1:91,1] = PR[GP1:90,1] + -1.522;
   1:  PR[GP1:91,2] = PR[GP1:90,2] + 32.359;
   1:  PR[GP1:91,3] = PR[GP1:90,3] + 67.830;
   1:L PR[91] 10mm/sec CNT100;
   1:  PR[GP1:91,1] = PR[GP1:90,1] + -2.200;
   1:  PR[GP1:91,2] = PR[GP1:90,2] + 32.516;
   1:L PR[91] 10mm/sec CNT100;
   1:  PR[GP1:91,1] = PR[GP1:90,1] + -2.797;
   1:  PR[GP1:91,2] = PR[GP1:90,2] + 32.938;
   1:L PR[91] 10mm/sec CNT100;
   1:  PR[GP1:91,1] = PR[GP1:90,1] + -3.099;
   1:  PR[GP1:91,2] = PR[GP1:90,2] + 33.096;
   1:L PR[91] 10mm/sec CNT100;
   1:  PR[GP1:91,1] = PR[GP1:90,1] + -3.520;
   1:  PR[GP1:91,2] = PR[GP1:90,2] + 33.231;
   1:L PR[91] 10mm/sec CNT100;
   1:  PR[GP1:91,1] = PR[GP1:90,1] + -15.736;
   1:  PR[GP1:91,2] = PR[GP1:90,2] + 37.455;
   1:L PR[91] 10mm/sec CNT100;
   1:  PR[GP1:91,1] = PR[GP1:90,1] + -16.672;
   1:  PR[GP1:91,2] = PR[GP1:90,2] + 37.577;
   1:L PR[91] 10mm/sec CNT100;
   1:  PR[GP1:91,1] = PR[GP1:90,1] + -17.837;
   1:  PR[GP1:91,2] = PR[GP1:90,2] + 37.537;
   1:L PR[91] 10mm/sec CNT100;
   1:  PR[GP1:91,1] = PR[GP1:90,1] + -29.665;
   1:  PR[GP1:91,2] = PR[GP1:90,2] + 37.478;
   1:L PR[91] 10mm/sec CNT100;
   1:  PR[GP1:91,1] = PR[GP1:90,1] + -31.249;
   1:  PR[GP1:91,2] = PR[GP1:90,2] + 37.136;
   1:L PR[91] 10mm/sec CNT100;
   1:  PR[GP1:91,1] = PR[GP1:90,1] + -33.039;
   1:  PR[GP1:91,2] = PR[GP1:90,2] + 36.427;
   1:L PR[91] 10mm/sec CNT100;
   1:  PR[GP1:91,1] = PR[GP1:90,1] + -42.783;
   1:  PR[GP1:91,2] = PR[GP1:90,2] + 32.967;
   1:L PR[91] 10mm/sec CNT100;
   1:  PR[GP1:91,1] = PR[GP1:90,1] + -44.722;
   1:  PR[GP1:91,2] = PR[GP1:90,2] + 31.760;
   1:L PR[91] 10mm/sec CNT100;
   1:  PR[GP1:91,1] = PR[GP1:90,1] + -46.644;
   1:  PR[GP1:91,2] = PR[GP1:90,2] + 30.053;
   1:L PR[91] 10mm/sec CNT100;
   1:  PR[GP1:91,1] = PR[GP1:90,1] + -53.515;
   1:  PR[GP1:91,2] = PR[GP1:90,2] + 24.493;
   1:L PR[91] 10mm/sec CNT100;
   1:  PR[GP1:91,1] = PR[GP1:90,1] + -55.197;
   1:  PR[GP1:91,2] = PR[GP1:90,2] + 22.303;
   1:L PR[91] 10mm/sec CNT100;
   1:  PR[GP1:91,1] = PR[GP1:90,1] + -56.634;
   1:  PR[GP1:91,2] = PR[GP1:90,2] + 19.515;
   1:L PR[91] 10mm/sec CNT100;
   1:  PR[GP1:91,1] = PR[GP1:90,1] + -60.582;
   1:  PR[GP1:91,2] = PR[GP1:90,2] + 12.919;
   1:L PR[91] 10mm/sec CNT100;
   1:  PR[GP1:91,1] = PR[GP1:90,1] + -61.433;
   1:  PR[GP1:91,2] = PR[GP1:90,2] + 10.034;
   1:L PR[91] 10mm/sec CNT100;
   1:  PR[GP1:91,1] = PR[GP1:90,1] + -61.717;
   1:  PR[GP1:91,2] = PR[GP1:90,2] + 6.920;
   1:L PR[91] 10mm/sec CNT100;
   1:  PR[GP1:91,1] = PR[GP1:90,1] + -62.999;
   1:  PR[GP1:91,2] = PR[GP1:90,2] + -0.032;
   1:L PR[91] 10mm/sec CNT100;
   1:  PR[GP1:91,1] = PR[GP1:90,1] + -62.720;
   1:  PR[GP1:91,2] = PR[GP1:90,2] + -3.121;
   1:L PR[91] 10mm/sec CNT100;
   1:  PR[GP1:91,1] = PR[GP1:90,1] + -61.440;
   1:  PR[GP1:91,2] = PR[GP1:90,2] + -10.019;
   1:L PR[91] 10mm/sec CNT100;
   1:  PR[GP1:91,1] = PR[GP1:90,1] + -60.575;
   1:  PR[GP1:91,2] = PR[GP1:90,2] + -12.950;
   1:L PR[91] 10mm/sec CNT100;
   1:  PR[GP1:91,1] = PR[GP1:90,1] + -59.176;
   1:  PR[GP1:91,2] = PR[GP1:90,2] + -15.694;
   1:L PR[91] 10mm/sec CNT100;
   1:  PR[GP1:91,1] = PR[GP1:90,1] + -55.205;
   1:  PR[GP1:91,2] = PR[GP1:90,2] + -22.300;
   1:L PR[91] 10mm/sec CNT100;
   1:  PR[GP1:91,1] = PR[GP1:90,1] + -53.502;
   1:  PR[GP1:91,2] = PR[GP1:90,2] + -24.518;
   1:L PR[91] 10mm/sec CNT100;
   1:  PR[GP1:91,1] = PR[GP1:90,1] + -51.585;
   1:  PR[GP1:91,2] = PR[GP1:90,2] + -26.238;
   1:L PR[91] 10mm/sec CNT100;
   1:  PR[GP1:91,1] = PR[GP1:90,1] + -44.726;
   1:  PR[GP1:91,2] = PR[GP1:90,2] + -31.765;
   1:L PR[91] 10mm/sec CNT100;
   1:  PR[GP1:91,1] = PR[GP1:90,1] + -42.765;
   1:  PR[GP1:91,2] = PR[GP1:90,2] + -32.987;
   1:L PR[91] 10mm/sec CNT100;
   1:  PR[GP1:91,1] = PR[GP1:90,1] + -40.841;
   1:  PR[GP1:91,2] = PR[GP1:90,2] + -33.759;
   1:L PR[91] 10mm/sec CNT100;
   1:  PR[GP1:91,1] = PR[GP1:90,1] + -31.246;
   1:  PR[GP1:91,2] = PR[GP1:90,2] + -37.145;
   1:L PR[91] 10mm/sec CNT100;
   1:  PR[GP1:91,1] = PR[GP1:90,1] + -29.642;
   1:  PR[GP1:91,2] = PR[GP1:90,2] + -37.491;
   1:L PR[91] 10mm/sec CNT100;
   1:  PR[GP1:91,1] = PR[GP1:90,1] + -28.177;
   1:  PR[GP1:91,2] = PR[GP1:90,2] + -37.547;
   1:L PR[91] 10mm/sec CNT100;
   1:  PR[GP1:91,1] = PR[GP1:90,1] + -16.662;
   1:  PR[GP1:91,2] = PR[GP1:90,2] + -37.584;
   1:L PR[91] 10mm/sec CNT100;
   1:  PR[GP1:91,1] = PR[GP1:90,1] + -15.709;
   1:  PR[GP1:91,2] = PR[GP1:90,2] + -37.459;
   1:L PR[91] 10mm/sec CNT100;
   1:  PR[GP1:91,1] = PR[GP1:90,1] + -14.878;
   1:  PR[GP1:91,2] = PR[GP1:90,2] + -37.195;
   1:L PR[91] 10mm/sec CNT100;
   1:  PR[GP1:91,1] = PR[GP1:90,1] + -3.085;
   1:  PR[GP1:91,2] = PR[GP1:90,2] + -33.097;
   1:L PR[91] 10mm/sec CNT100;
   1:  PR[GP1:91,1] = PR[GP1:90,1] + -2.789;
   1:  PR[GP1:91,2] = PR[GP1:90,2] + -32.942;
   1:L PR[91] 10mm/sec CNT100;
   1:  PR[GP1:91,1] = PR[GP1:90,1] + -2.156;
   1:  PR[GP1:91,2] = PR[GP1:90,2] + -32.482;
   1:L PR[91] 10mm/sec CNT100;
   1:  PR[GP1:91,1] = PR[GP1:90,1] + 0.738;
   1:  PR[GP1:91,2] = PR[GP1:90,2] + -32.366;
   1:L PR[91] 10mm/sec CNT100;
   1:  PR[GP1:91,1] = PR[GP1:90,1] + 2.335;
   1:  PR[GP1:91,2] = PR[GP1:90,2] + -32.025;
   1:L PR[91] 10mm/sec CNT100;
   1:  PR[GP1:91,1] = PR[GP1:90,1] + 2.871;
   1:  PR[GP1:91,2] = PR[GP1:90,2] + -32.457;
   1:L PR[91] 10mm/sec CNT100;
   1:  PR[GP1:91,1] = PR[GP1:90,1] + 3.076;
   1:  PR[GP1:91,2] = PR[GP1:90,2] + -32.559;
   1:L PR[91] 10mm/sec CNT100;
   1:  PR[GP1:91,1] = PR[GP1:90,1] + 3.603;
   1:  PR[GP1:91,2] = PR[GP1:90,2] + -32.942;
   1:L PR[91] 10mm/sec CNT100;
   1:  PR[GP1:91,1] = PR[GP1:90,1] + 3.890;
   1:  PR[GP1:91,2] = PR[GP1:90,2] + -33.092;
   1:L PR[91] 10mm/sec CNT100;
   1:  PR[GP1:91,1] = PR[GP1:90,1] + 4.302;
   1:  PR[GP1:91,2] = PR[GP1:90,2] + -33.224;
   1:L PR[91] 10mm/sec CNT100;
   1:  PR[GP1:91,1] = PR[GP1:90,1] + 16.534;
   1:  PR[GP1:91,2] = PR[GP1:90,2] + -37.459;
   1:L PR[91] 10mm/sec CNT100;
   1:  PR[GP1:91,1] = PR[GP1:90,1] + 17.468;
   1:  PR[GP1:91,2] = PR[GP1:90,2] + -37.582;
   1:L PR[91] 10mm/sec CNT100;
   1:  PR[GP1:91,1] = PR[GP1:90,1] + 18.626;
   1:  PR[GP1:91,2] = PR[GP1:90,2] + -37.543;
   1:L PR[91] 10mm/sec CNT100;
   1:  PR[GP1:91,1] = PR[GP1:90,1] + 30.460;
   1:  PR[GP1:91,2] = PR[GP1:90,2] + -37.491;
   1:L PR[91] 10mm/sec CNT100;
   1:  PR[GP1:91,1] = PR[GP1:90,1] + 32.041;
   1:  PR[GP1:91,2] = PR[GP1:90,2] + -37.151;
   1:L PR[91] 10mm/sec CNT100;
   1:  PR[GP1:91,1] = PR[GP1:90,1] + 33.833;
   1:  PR[GP1:91,2] = PR[GP1:90,2] + -36.445;
   1:L PR[91] 10mm/sec CNT100;
   1:  PR[GP1:91,1] = PR[GP1:90,1] + 43.584;
   1:  PR[GP1:91,2] = PR[GP1:90,2] + -32.989;
   1:L PR[91] 10mm/sec CNT100;
   1:  PR[GP1:91,1] = PR[GP1:90,1] + 45.510;
   1:  PR[GP1:91,2] = PR[GP1:90,2] + -31.795;
   1:L PR[91] 10mm/sec CNT100;
   1:  PR[GP1:91,1] = PR[GP1:90,1] + 47.421;
   1:  PR[GP1:91,2] = PR[GP1:90,2] + -30.103;
   1:L PR[91] 10mm/sec CNT100;
   1:  PR[GP1:91,1] = PR[GP1:90,1] + 54.297;
   1:  PR[GP1:91,2] = PR[GP1:90,2] + -24.537;
   1:L PR[91] 10mm/sec CNT100;
   1:  PR[GP1:91,1] = PR[GP1:90,1] + 55.997;
   1:  PR[GP1:91,2] = PR[GP1:90,2] + -22.330;
   1:L PR[91] 10mm/sec CNT100;
   1:  PR[GP1:91,1] = PR[GP1:90,1] + 57.438;
   1:  PR[GP1:91,2] = PR[GP1:90,2] + -19.565;
   1:L PR[91] 10mm/sec CNT100;
   1:  PR[GP1:91,1] = PR[GP1:90,1] + 61.389;
   1:  PR[GP1:91,2] = PR[GP1:90,2] + -12.981;
   1:L PR[91] 10mm/sec CNT100;
   1:  PR[GP1:91,1] = PR[GP1:90,1] + 62.238;
   1:  PR[GP1:91,2] = PR[GP1:90,2] + -10.140;
   1:L PR[91] 10mm/sec CNT100;
   1:  PR[GP1:91,1] = PR[GP1:90,1] + 62.537;
   1:  PR[GP1:91,2] = PR[GP1:90,2] + -6.940;
   1:L PR[91] 10mm/sec CNT100;
   1:  PR[GP1:91,1] = PR[GP1:90,1] + 63.820;
   1:  PR[GP1:91,2] = PR[GP1:90,2] + 0.023;
   1:L PR[91] 10mm/sec CNT100;
   1:  PR[GP1:91,1] = PR[GP1:90,1] + 63.526;
   1:  PR[GP1:91,2] = PR[GP1:90,2] + 3.199;
   1:L PR[91] 10mm/sec CNT100;
   1:  PR[GP1:91,1] = PR[GP1:90,1] + 62.247;
   1:  PR[GP1:91,2] = PR[GP1:90,2] + 10.103;
   1:L PR[91] 10mm/sec CNT100;
   1:  PR[GP1:91,1] = PR[GP1:90,1] + 61.385;
   1:  PR[GP1:91,2] = PR[GP1:90,2] + 12.989;
   1:L PR[91] 10mm/sec CNT100;
   1:  PR[GP1:91,1] = PR[GP1:90,1] + 59.981;
   1:  PR[GP1:91,2] = PR[GP1:90,2] + 15.710;
   1:L PR[91] 10mm/sec CNT100;
   1:  PR[GP1:91,1] = PR[GP1:90,1] + 56.012;
   1:  PR[GP1:91,2] = PR[GP1:90,2] + 22.302;
   1:L PR[91] 10mm/sec CNT100;
   1:  PR[GP1:91,1] = PR[GP1:90,1] + 54.291;
   1:  PR[GP1:91,2] = PR[GP1:90,2] + 24.536;
   1:L PR[91] 10mm/sec CNT100;
   1:  PR[GP1:91,1] = PR[GP1:90,1] + 52.384;
   1:  PR[GP1:91,2] = PR[GP1:90,2] + 26.242;
   1:L PR[91] 10mm/sec CNT100;
   1:  PR[GP1:91,1] = PR[GP1:90,1] + 45.529;
   1:  PR[GP1:91,2] = PR[GP1:90,2] + 31.775;
   1:L PR[91] 10mm/sec CNT100;
   1:  PR[GP1:91,1] = PR[GP1:90,1] + 43.582;
   1:  PR[GP1:91,2] = PR[GP1:90,2] + 32.982;
   1:L PR[91] 10mm/sec CNT100;
   1:  PR[GP1:91,1] = PR[GP1:90,1] + 41.655;
   1:  PR[GP1:91,2] = PR[GP1:90,2] + 33.751;
   1:L PR[91] 10mm/sec CNT100;
   1:  PR[GP1:91,1] = PR[GP1:90,1] + 32.065;
   1:  PR[GP1:91,2] = PR[GP1:90,2] + 37.137;
   1:L PR[91] 10mm/sec CNT100;
   1:  PR[GP1:91,1] = PR[GP1:90,1] + 30.464;
   1:  PR[GP1:91,2] = PR[GP1:90,2] + 37.482;
   1:L PR[91] 10mm/sec CNT100;
   1:  PR[GP1:91,1] = PR[GP1:90,1] + 29.006;
   1:  PR[GP1:91,2] = PR[GP1:90,2] + 37.537;
   1:L PR[91] 10mm/sec CNT100;
   1:  PR[GP1:91,1] = PR[GP1:90,1] + 17.496;
   1:  PR[GP1:91,2] = PR[GP1:90,2] + 37.577;
   1:L PR[91] 10mm/sec CNT100;
   1:  PR[GP1:91,1] = PR[GP1:90,1] + 16.545;
   1:  PR[GP1:91,2] = PR[GP1:90,2] + 37.452;
   1:L PR[91] 10mm/sec CNT100;
   1:  PR[GP1:91,1] = PR[GP1:90,1] + 15.712;
   1:  PR[GP1:91,2] = PR[GP1:90,2] + 37.187;
   1:L PR[91] 10mm/sec CNT100;
   1:  PR[GP1:91,1] = PR[GP1:90,1] + 3.916;
   1:  PR[GP1:91,2] = PR[GP1:90,2] + 33.097;
   1:L PR[91] 10mm/sec CNT100;
   1:  PR[GP1:91,1] = PR[GP1:90,1] + 3.611;
   1:  PR[GP1:91,2] = PR[GP1:90,2] + 32.938;
   1:L PR[91] 10mm/sec CNT100;
   1:  PR[GP1:91,1] = PR[GP1:90,1] + 3.379;
   1:  PR[GP1:91,2] = PR[GP1:90,2] + 32.775;
   1:L PR[91] 10mm/sec CNT100;
   1:  PR[GP1:91,1] = PR[GP1:90,1] + 3.386;
   1:  PR[GP1:91,2] = PR[GP1:90,2] + 32.645;
   1:L PR[91] 10mm/sec CNT100;
   1:  PR[GP1:91,1] = PR[GP1:90,1] + 2.307;
   1:  PR[GP1:91,2] = PR[GP1:90,2] + 32.044;
   1:L PR[91] 10mm/sec CNT100;
   1:  PR[GP1:91,1] = PR[GP1:90,1] + -1.850;
   1:  PR[GP1:91,2] = PR[GP1:90,2] + 32.921;
   1:  PR[GP1:91,3] = PR[GP1:90,3] + 69.160;
   1:L PR[91] 10mm/sec CNT100;
   1:  PR[GP1:91,1] = PR[GP1:90,1] + -2.123;
   1:  PR[GP1:91,2] = PR[GP1:90,2] + 32.985;
   1:L PR[91] 10mm/sec CNT100;
   1:  PR[GP1:91,1] = PR[GP1:90,1] + -2.382;
   1:  PR[GP1:91,2] = PR[GP1:90,2] + 33.148;
   1:L PR[91] 10mm/sec CNT100;
   1:  PR[GP1:91,1] = PR[GP1:90,1] + -15.303;
   1:  PR[GP1:91,2] = PR[GP1:90,2] + 37.612;
   1:L PR[91] 10mm/sec CNT100;
   1:  PR[GP1:91,1] = PR[GP1:90,1] + -15.906;
   1:  PR[GP1:91,2] = PR[GP1:90,2] + 37.691;
   1:L PR[91] 10mm/sec CNT100;
   1:  PR[GP1:91,1] = PR[GP1:90,1] + -16.685;
   1:  PR[GP1:91,2] = PR[GP1:90,2] + 37.664;
   1:L PR[91] 10mm/sec CNT100;
   1:  PR[GP1:91,1] = PR[GP1:90,1] + -29.256;
   1:  PR[GP1:91,2] = PR[GP1:90,2] + 37.601;
   1:L PR[91] 10mm/sec CNT100;
   1:  PR[GP1:91,1] = PR[GP1:90,1] + -30.495;
   1:  PR[GP1:91,2] = PR[GP1:90,2] + 37.334;
   1:L PR[91] 10mm/sec CNT100;
   1:  PR[GP1:91,1] = PR[GP1:90,1] + -31.914;
   1:  PR[GP1:91,2] = PR[GP1:90,2] + 36.772;
   1:L PR[91] 10mm/sec CNT100;
   1:  PR[GP1:91,1] = PR[GP1:90,1] + -42.383;
   1:  PR[GP1:91,2] = PR[GP1:90,2] + 33.054;
   1:L PR[91] 10mm/sec CNT100;
   1:  PR[GP1:91,1] = PR[GP1:90,1] + -44.013;
   1:  PR[GP1:91,2] = PR[GP1:90,2] + 32.039;
   1:L PR[91] 10mm/sec CNT100;
   1:  PR[GP1:91,1] = PR[GP1:90,1] + -45.640;
   1:  PR[GP1:91,2] = PR[GP1:90,2] + 30.595;
   1:L PR[91] 10mm/sec CNT100;
   1:  PR[GP1:91,1] = PR[GP1:90,1] + -53.115;
   1:  PR[GP1:91,2] = PR[GP1:90,2] + 24.546;
   1:L PR[91] 10mm/sec CNT100;
   1:  PR[GP1:91,1] = PR[GP1:90,1] + -54.576;
   1:  PR[GP1:91,2] = PR[GP1:90,2] + 22.643;
   1:L PR[91] 10mm/sec CNT100;
   1:  PR[GP1:91,1] = PR[GP1:90,1] + -55.831;
   1:  PR[GP1:91,2] = PR[GP1:90,2] + 20.209;
   1:L PR[91] 10mm/sec CNT100;
   1:  PR[GP1:91,1] = PR[GP1:90,1] + -60.174;
   1:  PR[GP1:91,2] = PR[GP1:90,2] + 12.954;
   1:L PR[91] 10mm/sec CNT100;
   1:  PR[GP1:91,1] = PR[GP1:90,1] + -60.924;
   1:  PR[GP1:91,2] = PR[GP1:90,2] + 10.409;
   1:L PR[91] 10mm/sec CNT100;
   1:  PR[GP1:91,1] = PR[GP1:90,1] + -61.177;
   1:  PR[GP1:91,2] = PR[GP1:90,2] + 7.649;
   1:L PR[91] 10mm/sec CNT100;
   1:  PR[GP1:91,1] = PR[GP1:90,1] + -62.593;
   1:  PR[GP1:91,2] = PR[GP1:90,2] + -0.032;
   1:L PR[91] 10mm/sec CNT100;
   1:  PR[GP1:91,1] = PR[GP1:90,1] + -62.345;
   1:  PR[GP1:91,2] = PR[GP1:90,2] + -2.780;
   1:L PR[91] 10mm/sec CNT100;
   1:  PR[GP1:91,1] = PR[GP1:90,1] + -60.931;
   1:  PR[GP1:91,2] = PR[GP1:90,2] + -10.393;
   1:L PR[91] 10mm/sec CNT100;
   1:  PR[GP1:91,1] = PR[GP1:90,1] + -60.168;
   1:  PR[GP1:91,2] = PR[GP1:90,2] + -12.985;
   1:L PR[91] 10mm/sec CNT100;
   1:  PR[GP1:91,1] = PR[GP1:90,1] + -58.930;
   1:  PR[GP1:91,2] = PR[GP1:90,2] + -15.411;
   1:L PR[91] 10mm/sec CNT100;
   1:  PR[GP1:91,1] = PR[GP1:90,1] + -54.585;
   1:  PR[GP1:91,2] = PR[GP1:90,2] + -22.641;
   1:L PR[91] 10mm/sec CNT100;
   1:  PR[GP1:91,1] = PR[GP1:90,1] + -53.102;
   1:  PR[GP1:91,2] = PR[GP1:90,2] + -24.571;
   1:L PR[91] 10mm/sec CNT100;
   1:  PR[GP1:91,1] = PR[GP1:90,1] + -51.432;
   1:  PR[GP1:91,2] = PR[GP1:90,2] + -26.069;
   1:L PR[91] 10mm/sec CNT100;
   1:  PR[GP1:91,1] = PR[GP1:90,1] + -44.017;
   1:  PR[GP1:91,2] = PR[GP1:90,2] + -32.045;
   1:L PR[91] 10mm/sec CNT100;
   1:  PR[GP1:91,1] = PR[GP1:90,1] + -42.364;
   1:  PR[GP1:91,2] = PR[GP1:90,2] + -33.075;
   1:L PR[91] 10mm/sec CNT100;
   1:  PR[GP1:91,1] = PR[GP1:90,1] + -40.741;
   1:  PR[GP1:91,2] = PR[GP1:90,2] + -33.726;
   1:L PR[91] 10mm/sec CNT100;
   1:  PR[GP1:91,1] = PR[GP1:90,1] + -30.492;
   1:  PR[GP1:91,2] = PR[GP1:90,2] + -37.343;
   1:L PR[91] 10mm/sec CNT100;
   1:  PR[GP1:91,1] = PR[GP1:90,1] + -29.231;
   1:  PR[GP1:91,2] = PR[GP1:90,2] + -37.614;
   1:L PR[91] 10mm/sec CNT100;
   1:  PR[GP1:91,1] = PR[GP1:90,1] + -28.078;
   1:  PR[GP1:91,2] = PR[GP1:90,2] + -37.659;
   1:L PR[91] 10mm/sec CNT100;
   1:  PR[GP1:91,1] = PR[GP1:90,1] + -15.894;
   1:  PR[GP1:91,2] = PR[GP1:90,2] + -37.697;
   1:L PR[91] 10mm/sec CNT100;
   1:  PR[GP1:91,1] = PR[GP1:90,1] + -15.276;
   1:  PR[GP1:91,2] = PR[GP1:90,2] + -37.617;
   1:L PR[91] 10mm/sec CNT100;
   1:  PR[GP1:91,1] = PR[GP1:90,1] + -14.729;
   1:  PR[GP1:91,2] = PR[GP1:90,2] + -37.443;
   1:L PR[91] 10mm/sec CNT100;
   1:  PR[GP1:91,1] = PR[GP1:90,1] + -2.364;
   1:  PR[GP1:91,2] = PR[GP1:90,2] + -33.146;
   1:L PR[91] 10mm/sec CNT100;
   1:  PR[GP1:91,1] = PR[GP1:90,1] + -2.076;
   1:  PR[GP1:91,2] = PR[GP1:90,2] + -32.961;
   1:L PR[91] 10mm/sec CNT100;
   1:  PR[GP1:91,1] = PR[GP1:90,1] + 1.100;
   1:  PR[GP1:91,2] = PR[GP1:90,2] + -32.834;
   1:L PR[91] 10mm/sec CNT100;
   1:  PR[GP1:91,1] = PR[GP1:90,1] + 2.401;
   1:  PR[GP1:91,2] = PR[GP1:90,2] + -32.556;
   1:L PR[91] 10mm/sec CNT100;
   1:  PR[GP1:91,1] = PR[GP1:90,1] + 2.997;
   1:  PR[GP1:91,2] = PR[GP1:90,2] + -33.036;
   1:L PR[91] 10mm/sec CNT100;
   1:  PR[GP1:91,1] = PR[GP1:90,1] + 3.170;
   1:  PR[GP1:91,2] = PR[GP1:90,2] + -33.142;
   1:L PR[91] 10mm/sec CNT100;
   1:  PR[GP1:91,1] = PR[GP1:90,1] + 16.100;
   1:  PR[GP1:91,2] = PR[GP1:90,2] + -37.616;
   1:L PR[91] 10mm/sec CNT100;
   1:  PR[GP1:91,1] = PR[GP1:90,1] + 16.701;
   1:  PR[GP1:91,2] = PR[GP1:90,2] + -37.695;
   1:L PR[91] 10mm/sec CNT100;
   1:  PR[GP1:91,1] = PR[GP1:90,1] + 17.476;
   1:  PR[GP1:91,2] = PR[GP1:90,2] + -37.669;
   1:L PR[91] 10mm/sec CNT100;
   1:  PR[GP1:91,1] = PR[GP1:90,1] + 30.052;
   1:  PR[GP1:91,2] = PR[GP1:90,2] + -37.614;
   1:L PR[91] 10mm/sec CNT100;
   1:  PR[GP1:91,1] = PR[GP1:90,1] + 31.289;
   1:  PR[GP1:91,2] = PR[GP1:90,2] + -37.348;
   1:L PR[91] 10mm/sec CNT100;
   1:  PR[GP1:91,1] = PR[GP1:90,1] + 32.709;
   1:  PR[GP1:91,2] = PR[GP1:90,2] + -36.788;
   1:L PR[91] 10mm/sec CNT100;
   1:  PR[GP1:91,1] = PR[GP1:90,1] + 43.185;
   1:  PR[GP1:91,2] = PR[GP1:90,2] + -33.076;
   1:L PR[91] 10mm/sec CNT100;
   1:  PR[GP1:91,1] = PR[GP1:90,1] + 44.804;
   1:  PR[GP1:91,2] = PR[GP1:90,2] + -32.072;
   1:L PR[91] 10mm/sec CNT100;
   1:  PR[GP1:91,1] = PR[GP1:90,1] + 46.421;
   1:  PR[GP1:91,2] = PR[GP1:90,2] + -30.640;
   1:L PR[91] 10mm/sec CNT100;
   1:  PR[GP1:91,1] = PR[GP1:90,1] + 53.901;
   1:  PR[GP1:91,2] = PR[GP1:90,2] + -24.586;
   1:L PR[91] 10mm/sec CNT100;
   1:  PR[GP1:91,1] = PR[GP1:90,1] + 55.378;
   1:  PR[GP1:91,2] = PR[GP1:90,2] + -22.667;
   1:L PR[91] 10mm/sec CNT100;
   1:  PR[GP1:91,1] = PR[GP1:90,1] + 56.636;
   1:  PR[GP1:91,2] = PR[GP1:90,2] + -20.253;
   1:L PR[91] 10mm/sec CNT100;
   1:  PR[GP1:91,1] = PR[GP1:90,1] + 60.983;
   1:  PR[GP1:91,2] = PR[GP1:90,2] + -13.012;
   1:L PR[91] 10mm/sec CNT100;
   1:  PR[GP1:91,1] = PR[GP1:90,1] + 61.732;
   1:  PR[GP1:91,2] = PR[GP1:90,2] + -10.506;
   1:L PR[91] 10mm/sec CNT100;
   1:  PR[GP1:91,1] = PR[GP1:90,1] + 61.997;
   1:  PR[GP1:91,2] = PR[GP1:90,2] + -7.670;
   1:L PR[91] 10mm/sec CNT100;
   1:  PR[GP1:91,1] = PR[GP1:90,1] + 63.413;
   1:  PR[GP1:91,2] = PR[GP1:90,2] + 0.023;
   1:L PR[91] 10mm/sec CNT100;
   1:  PR[GP1:91,1] = PR[GP1:90,1] + 63.153;
   1:  PR[GP1:91,2] = PR[GP1:90,2] + 2.849;
   1:L PR[91] 10mm/sec CNT100;
   1:  PR[GP1:91,1] = PR[GP1:90,1] + 61.740;
   1:  PR[GP1:91,2] = PR[GP1:90,2] + 10.468;
   1:L PR[91] 10mm/sec CNT100;
   1:  PR[GP1:91,1] = PR[GP1:90,1] + 60.978;
   1:  PR[GP1:91,2] = PR[GP1:90,2] + 13.019;
   1:L PR[91] 10mm/sec CNT100;
   1:  PR[GP1:91,1] = PR[GP1:90,1] + 59.736;
   1:  PR[GP1:91,2] = PR[GP1:90,2] + 15.426;
   1:L PR[91] 10mm/sec CNT100;
   1:  PR[GP1:91,1] = PR[GP1:90,1] + 55.393;
   1:  PR[GP1:91,2] = PR[GP1:90,2] + 22.640;
   1:L PR[91] 10mm/sec CNT100;
   1:  PR[GP1:91,1] = PR[GP1:90,1] + 53.895;
   1:  PR[GP1:91,2] = PR[GP1:90,2] + 24.584;
   1:L PR[91] 10mm/sec CNT100;
   1:  PR[GP1:91,1] = PR[GP1:90,1] + 52.234;
   1:  PR[GP1:91,2] = PR[GP1:90,2] + 26.070;
   1:L PR[91] 10mm/sec CNT100;
   1:  PR[GP1:91,1] = PR[GP1:90,1] + 44.824;
   1:  PR[GP1:91,2] = PR[GP1:90,2] + 32.051;
   1:L PR[91] 10mm/sec CNT100;
   1:  PR[GP1:91,1] = PR[GP1:90,1] + 43.183;
   1:  PR[GP1:91,2] = PR[GP1:90,2] + 33.068;
   1:L PR[91] 10mm/sec CNT100;
   1:  PR[GP1:91,1] = PR[GP1:90,1] + 41.558;
   1:  PR[GP1:91,2] = PR[GP1:90,2] + 33.718;
   1:L PR[91] 10mm/sec CNT100;
   1:  PR[GP1:91,1] = PR[GP1:90,1] + 31.314;
   1:  PR[GP1:91,2] = PR[GP1:90,2] + 37.334;
   1:L PR[91] 10mm/sec CNT100;
   1:  PR[GP1:91,1] = PR[GP1:90,1] + 30.056;
   1:  PR[GP1:91,2] = PR[GP1:90,2] + 37.605;
   1:L PR[91] 10mm/sec CNT100;
   1:  PR[GP1:91,1] = PR[GP1:90,1] + 28.908;
   1:  PR[GP1:91,2] = PR[GP1:90,2] + 37.648;
   1:L PR[91] 10mm/sec CNT100;
   1:  PR[GP1:91,1] = PR[GP1:90,1] + 16.730;
   1:  PR[GP1:91,2] = PR[GP1:90,2] + 37.691;
   1:L PR[91] 10mm/sec CNT100;
   1:  PR[GP1:91,1] = PR[GP1:90,1] + 16.112;
   1:  PR[GP1:91,2] = PR[GP1:90,2] + 37.610;
   1:L PR[91] 10mm/sec CNT100;
   1:  PR[GP1:91,1] = PR[GP1:90,1] + 15.564;
   1:  PR[GP1:91,2] = PR[GP1:90,2] + 37.435;
   1:L PR[91] 10mm/sec CNT100;
   1:  PR[GP1:91,1] = PR[GP1:90,1] + 3.321;
   1:  PR[GP1:91,2] = PR[GP1:90,2] + 33.191;
   1:L PR[91] 10mm/sec CNT100;
   1:  PR[GP1:91,1] = PR[GP1:90,1] + 3.326;
   1:  PR[GP1:91,2] = PR[GP1:90,2] + 33.105;
   1:L PR[91] 10mm/sec CNT100;
   1:  PR[GP1:91,1] = PR[GP1:90,1] + 2.372;
   1:  PR[GP1:91,2] = PR[GP1:90,2] + 32.575;
   1:L PR[91] 10mm/sec CNT100;
   1:  PR[GP1:91,1] = PR[GP1:90,1] + -1.038;
   1:  PR[GP1:91,2] = PR[GP1:90,2] + 33.390;
   1:  PR[GP1:91,3] = PR[GP1:90,3] + 70.490;
   1:L PR[91] 10mm/sec CNT100;
   1:  PR[GP1:91,1] = PR[GP1:90,1] + -1.923;
   1:  PR[GP1:91,2] = PR[GP1:90,2] + 33.385;
   1:L PR[91] 10mm/sec CNT100;
   1:  PR[GP1:91,1] = PR[GP1:90,1] + -6.628;
   1:  PR[GP1:91,2] = PR[GP1:90,2] + 34.920;
   1:L PR[91] 10mm/sec CNT100;
   1:  PR[GP1:91,1] = PR[GP1:90,1] + -14.871;
   1:  PR[GP1:91,2] = PR[GP1:90,2] + 37.770;
   1:L PR[91] 10mm/sec CNT100;
   1:  PR[GP1:91,1] = PR[GP1:90,1] + -15.139;
   1:  PR[GP1:91,2] = PR[GP1:90,2] + 37.805;
   1:L PR[91] 10mm/sec CNT100;
   1:  PR[GP1:91,1] = PR[GP1:90,1] + -15.534;
   1:  PR[GP1:91,2] = PR[GP1:90,2] + 37.791;
   1:L PR[91] 10mm/sec CNT100;
   1:  PR[GP1:91,1] = PR[GP1:90,1] + -28.846;
   1:  PR[GP1:91,2] = PR[GP1:90,2] + 37.724;
   1:L PR[91] 10mm/sec CNT100;
   1:  PR[GP1:91,1] = PR[GP1:90,1] + -29.742;
   1:  PR[GP1:91,2] = PR[GP1:90,2] + 37.531;
   1:L PR[91] 10mm/sec CNT100;
   1:  PR[GP1:91,1] = PR[GP1:90,1] + -30.790;
   1:  PR[GP1:91,2] = PR[GP1:90,2] + 37.116;
   1:L PR[91] 10mm/sec CNT100;
   1:  PR[GP1:91,1] = PR[GP1:90,1] + -41.983;
   1:  PR[GP1:91,2] = PR[GP1:90,2] + 33.142;
   1:L PR[91] 10mm/sec CNT100;
   1:  PR[GP1:91,1] = PR[GP1:90,1] + -43.305;
   1:  PR[GP1:91,2] = PR[GP1:90,2] + 32.318;
   1:L PR[91] 10mm/sec CNT100;
   1:  PR[GP1:91,1] = PR[GP1:90,1] + -44.636;
   1:  PR[GP1:91,2] = PR[GP1:90,2] + 31.136;
   1:L PR[91] 10mm/sec CNT100;
   1:  PR[GP1:91,1] = PR[GP1:90,1] + -52.715;
   1:  PR[GP1:91,2] = PR[GP1:90,2] + 24.599;
   1:L PR[91] 10mm/sec CNT100;
   1:  PR[GP1:91,1] = PR[GP1:90,1] + -53.956;
   1:  PR[GP1:91,2] = PR[GP1:90,2] + 22.983;
   1:L PR[91] 10mm/sec CNT100;
   1:  PR[GP1:91,1] = PR[GP1:90,1] + -55.028;
   1:  PR[GP1:91,2] = PR[GP1:90,2] + 20.903;
   1:L PR[91] 10mm/sec CNT100;
   1:  PR[GP1:91,1] = PR[GP1:90,1] + -59.766;
   1:  PR[GP1:91,2] = PR[GP1:90,2] + 12.988;
   1:L PR[91] 10mm/sec CNT100;
   1:  PR[GP1:91,1] = PR[GP1:90,1] + -60.416;
   1:  PR[GP1:91,2] = PR[GP1:90,2] + 10.783;
   1:L PR[91] 10mm/sec CNT100;
   1:  PR[GP1:91,1] = PR[GP1:90,1] + -60.636;
   1:  PR[GP1:91,2] = PR[GP1:90,2] + 8.378;
   1:L PR[91] 10mm/sec CNT100;
   1:  PR[GP1:91,1] = PR[GP1:90,1] + -62.187;
   1:  PR[GP1:91,2] = PR[GP1:90,2] + -0.032;
   1:L PR[91] 10mm/sec CNT100;
   1:  PR[GP1:91,1] = PR[GP1:90,1] + -61.969;
   1:  PR[GP1:91,2] = PR[GP1:90,2] + -2.439;
   1:L PR[91] 10mm/sec CNT100;
   1:  PR[GP1:91,1] = PR[GP1:90,1] + -60.423;
   1:  PR[GP1:91,2] = PR[GP1:90,2] + -10.768;
   1:L PR[91] 10mm/sec CNT100;
   1:  PR[GP1:91,1] = PR[GP1:90,1] + -59.760;
   1:  PR[GP1:91,2] = PR[GP1:90,2] + -13.019;
   1:L PR[91] 10mm/sec CNT100;
   1:  PR[GP1:91,1] = PR[GP1:90,1] + -58.684;
   1:  PR[GP1:91,2] = PR[GP1:90,2] + -15.128;
   1:L PR[91] 10mm/sec CNT100;
   1:  PR[GP1:91,1] = PR[GP1:90,1] + -53.964;
   1:  PR[GP1:91,2] = PR[GP1:90,2] + -22.981;
   1:L PR[91] 10mm/sec CNT100;
   1:  PR[GP1:91,1] = PR[GP1:90,1] + -52.701;
   1:  PR[GP1:91,2] = PR[GP1:90,2] + -24.624;
   1:L PR[91] 10mm/sec CNT100;
   1:  PR[GP1:91,1] = PR[GP1:90,1] + -51.279;
   1:  PR[GP1:91,2] = PR[GP1:90,2] + -25.901;
   1:L PR[91] 10mm/sec CNT100;
   1:  PR[GP1:91,1] = PR[GP1:90,1] + -43.308;
   1:  PR[GP1:91,2] = PR[GP1:90,2] + -32.325;
   1:L PR[91] 10mm/sec CNT100;
   1:  PR[GP1:91,1] = PR[GP1:90,1] + -41.964;
   1:  PR[GP1:91,2] = PR[GP1:90,2] + -33.162;
   1:L PR[91] 10mm/sec CNT100;
   1:  PR[GP1:91,1] = PR[GP1:90,1] + -40.642;
   1:  PR[GP1:91,2] = PR[GP1:90,2] + -33.693;
   1:L PR[91] 10mm/sec CNT100;
   1:  PR[GP1:91,1] = PR[GP1:90,1] + -29.737;
   1:  PR[GP1:91,2] = PR[GP1:90,2] + -37.540;
   1:L PR[91] 10mm/sec CNT100;
   1:  PR[GP1:91,1] = PR[GP1:90,1] + -28.821;
   1:  PR[GP1:91,2] = PR[GP1:90,2] + -37.738;
   1:L PR[91] 10mm/sec CNT100;
   1:  PR[GP1:91,1] = PR[GP1:90,1] + -27.978;
   1:  PR[GP1:91,2] = PR[GP1:90,2] + -37.770;
   1:L PR[91] 10mm/sec CNT100;
   1:  PR[GP1:91,1] = PR[GP1:90,1] + -15.126;
   1:  PR[GP1:91,2] = PR[GP1:90,2] + -37.811;
   1:L PR[91] 10mm/sec CNT100;
   1:  PR[GP1:91,1] = PR[GP1:90,1] + -14.842;
   1:  PR[GP1:91,2] = PR[GP1:90,2] + -37.774;
   1:L PR[91] 10mm/sec CNT100;
   1:  PR[GP1:91,1] = PR[GP1:90,1] + -14.580;
   1:  PR[GP1:91,2] = PR[GP1:90,2] + -37.690;
   1:L PR[91] 10mm/sec CNT100;
   1:  PR[GP1:91,1] = PR[GP1:90,1] + -6.762;
   1:  PR[GP1:91,2] = PR[GP1:90,2] + -34.974;
   1:L PR[91] 10mm/sec CNT100;
